	OUT_EV_HP => EV104,
	OUT_EV_LP => EV102,
(*	OUT_EV_LNK=> ,*)
	OUT_KEY   => KEY_PP2,
	OUT_THR   => THR_PP2
);
(*Link*)
EV107 := fbPP1.OUT_EV_LNK OR fbPP2.OUT_EV_LNK;  (******ANADIR si hace falta para la vibracion**************)

(*Alarms*)
Mute   := Mute   AND S101.AlLow AND S102.AlLow;
Bypass := Bypass AND (NOT S101.AlMax OR NOT S102.AlMax);
Buzzer := TANK.Enable AND (S101.AlHig OR S102.AlHig OR S101.AlMax OR S102.AlMax) AND NOT MUTE;

(*THROTTLE CALIBRATION*)
IF Calib1 THEN
	Calib2 := FALSE;

	CalThr := CalThr + CalInc;
	IF CalThr > CalMax THEN CalThr := CalMax; END_IF

	THR_PP1 := CalThr;
	THR_PP2 := 0.0;

	KEY_PP1 := TRUE;
	KEY_PP2 := TRUE;

	EV101 := FALSE;
	EV102 := FALSE;
	EV103 := FALSE;
	EV104 := FALSE;
ELSE
	CalThr := 0.0;
END_IF

IF Calib2 THEN
	Calib1 := FALSE;

	CalThr := CalThr + CalInc;
	IF CalThr > CalMax THEN CalThr := CalMax; END_IF

	THR_PP1 := 0.0;
	THR_PP2 := CalThr;

	KEY_PP1 := TRUE;
	KEY_PP2 := TRUE;

	EV101 := FALSE;
	EV102 := FALSE;
	EV103 := FALSE;
	EV104 := FALSE;
ELSE
	CalThr := 0.0;
END_IF
END_PROGRAM

(* POU FB/FB_POWERPACK, ST *)
FUNCTION_BLOCK FB_POWERPACK
VAR_INPUT
	Enable : BOOL;

	IN_HP : BOOL;
	IN_LP : BOOL;
END_VAR
VAR_IN_OUT
	HP_P : ST_SENSOR_BAR;
	LP_P : ST_SENSOR_BAR;
	CFG  : ST_POWERPACK_CFG;
END_VAR
VAR_OUTPUT
	OUT_EV_HP : BOOL;
	OUT_EV_LP : BOOL;
	OUT_EV_LNK: BOOL;
	OUT_KEY   : BOOL;
	OUT_THR   : REAL;
END_VAR
VAR
	State    : WORD;
	Hyst_Cnt : REAL;
	Hyst_ON  : BOOL;
	Thr_Cnt  : REAL;

END_VAR
IF NOT Enable THEN
	OUT_EV_HP  := FALSE;
	OUT_EV_LP  := FALSE;
	OUT_EV_LNK := FALSE;
	OUT_KEY    := FALSE;
	OUT_THR    := 0.0;

	State := 0;
	RETURN;
END_IF

IF LP_P.AlMax THEN IN_LP := FALSE; END_IF
IF HP_P.AlMax THEN IN_HP := FALSE; END_IF

CASE State OF
0: (*Init*)
	IF IN_LP AND IN_HP THEN
		OUT_EV_HP := TRUE;
		OUT_EV_LP := TRUE;
		OUT_EV_LNK:= FALSE;
		OUT_KEY   := TRUE;

		State := 30;

	ELSIF IN_LP THEN
		OUT_EV_HP := TRUE; (*Only LP Go with HP too*)
		OUT_EV_LP := TRUE;
		OUT_EV_LNK:= TRUE; (*Only LP Go with HP too*)
		OUT_KEY   := TRUE;

		Hyst_cnt := CFG.Hyst_TM + CFG.Cycle;
		State    := 10;

	ELSIF IN_HP THEN
		OUT_EV_HP := TRUE;
		OUT_EV_LP := FALSE;
		OUT_EV_LNK:= FALSE;
		OUT_KEY   := TRUE;

		State    := 20;

	ELSE
		OUT_EV_HP := FALSE;
		OUT_EV_LP := FALSE;
		OUT_EV_LNK:= FALSE;
		OUT_KEY   := FALSE;

	END_IF

	Thr_Cnt := 0.0;

10: (*LOW PRESS*)
	IF NOT IN_LP AND NOT IN_HP THEN
		OUT_EV_HP := FALSE;
		OUT_EV_LP := FALSE;
		OUT_EV_LNK:= FALSE;
		OUT_KEY   := FALSE;

		State := 0;

	ELSIF NOT IN_LP THEN (*Go to HP*)
		OUT_EV_HP := TRUE;
		OUT_EV_LP := FALSE;
		OUT_EV_LNK:= FALSE;

		State := 20;

	ELSIF IN_HP THEN
		OUT_EV_HP := TRUE;
		OUT_EV_LP := TRUE;
		OUT_EV_LNK:= FALSE;

		State := 30;

	ELSE
		IF Hyst_Cnt > CFG.Hyst_TM THEN
			Hyst_ON := TRUE;
		ELSE
			Hyst_ON  := FALSE;
			Hyst_Cnt := Hyst_Cnt + CFG.Cycle;
		END_IF

		IF LP_P.Bar > CFG.Hyst_HP AND Hyst_ON OR LP_P.Err THEN
			OUT_EV_HP  := FALSE;
			OUT_EV_LP  := TRUE;
			OUT_EV_LNK := FALSE;

			Hyst_cnt   := 0.0;

		ELSIF LP_P.Bar < CFG.Hyst_LP AND Hyst_ON THEN
			OUT_EV_HP  := TRUE; (*Only LP Go with HP too*)
			OUT_EV_LP  := TRUE;
			OUT_EV_LNK := TRUE; (*Only LP Go with HP too*)

			Hyst_cnt := 0.0;

		END_IF

	END_IF

20: (*HIGH PRESS*)
	IF NOT IN_LP AND NOT IN_HP THEN
		OUT_EV_HP := FALSE;
		OUT_EV_LP := FALSE;
		OUT_EV_LNK:= FALSE;
		OUT_KEY   := FALSE;

		State     := 0;

	ELSIF NOT IN_HP THEN
		OUT_EV_HP  := TRUE; (*Only LP Go with HP too*)
		OUT_EV_LP  := TRUE;
		OUT_EV_LNK := TRUE; (*Only LP Go with HP too*)

		Hyst_cnt := CFG.Hyst_TM + CFG.Cycle;
		State    := 10;

	ELSIF IN_LP THEN
		OUT_EV_HP := TRUE;
		OUT_EV_LP := TRUE;
		OUT_EV_LNK:= FALSE;

		State := 30;

	ELSE
		OUT_EV_HP := TRUE;
		OUT_EV_LP := FALSE;
		OUT_EV_LNK:= FALSE;

	END_IF

30: (*HP & LP*)
	IF NOT IN_LP AND NOT IN_HP THEN
		OUT_EV_HP := FALSE;
		OUT_EV_LP := FALSE;
		OUT_EV_LNK:= FALSE;
		OUT_KEY   := FALSE;

		State     := 0;

	ELSIF NOT IN_HP THEN (*Go to LP*)
		OUT_EV_HP  := TRUE; (*Only LP Go with HP too*)
		OUT_EV_LP  := TRUE;
		OUT_EV_LNK := TRUE; (*Only LP Go with HP too*)

		Hyst_cnt := CFG.Hyst_TM + CFG.Cycle;
		State    := 10;

	ELSIF NOT IN_LP THEN (*Go to HP*)
		OUT_EV_HP := TRUE;
		OUT_EV_LP := FALSE;
		OUT_EV_LNK:= FALSE;

		State := 20;

	ELSE
		OUT_EV_HP := TRUE;
		OUT_EV_LP := TRUE;
		OUT_EV_LNK:= FALSE;

	END_IF

END_CASE

IF OUT_KEY THEN
	IF Thr_Cnt > 0.2 THEN
		IF OUT_EV_HP AND OUT_EV_LP THEN
			OUT_Thr := MAX(CFG.Thr_HP,CFG.Thr_LP);
		ELSIF OUT_EV_LP THEN
			OUT_Thr := CFG.Thr_LP;
		ELSE
			OUT_Thr := CFG.Thr_HP;
		END_IF

	ELSE
		Thr_Cnt := Thr_Cnt + CFG.Cycle;
		OUT_Thr := 0.0;
	END_IF

ELSE
	OUT_THR := 0.0;

END_IF
END_FUNCTION_BLOCK

(* POU TOFARO, ST *)
PROGRAM TOFARO
VAR CONSTANT
	UDP_BUF_SIZE  : WORD := 4096;

END_VAR
VAR
	fbUdpSend        : FB_UDP_SEND;
	fbUdpRecv        : FB_UDP_RECV;
	fbSocketCloseAll : FB_SocketCloseAll;
    bCloseAll 	     : BOOL := TRUE;

	Send_Id          : DWORD;
	Send_NumberOfVars: WORD;
	Send_Offset      : WORD;
	Send_Buffer      : ARRAY[0..UDP_BUF_SIZE] OF BYTE;

	AuxVar : REAL;

	Recv_Id          : DWORD;
	Recv_NumberOfVars: WORD;
	Recv_Offset      : WORD;
	Recv_Buffer      : ARRAY[0..UDP_BUF_SIZE] OF BYTE;
	Recv_ToggleOLD   : BOOL;
	Recv_OldId       : DWORD;
	NoRecv_Cnt       : REAL;
	Recv_Live        : BOOL;

	rBar1 : REAL;
	rBar2 : REAL;
	rHeel : REAL;

	rRunP : REAL;
	rPriP : REAL;
	rMain : REAL;
	rRunS : REAL;
	rPriS : REAL;
	rSecP : REAL;
	rSecS : REAL;



END_VAR
(*UDP STREAMING*)
IF bCloseAll THEN (*On PLC reset or program download close all old connections *)
	bCloseAll := FALSE;
	fbUdpSend( bEnable:= FALSE );
	fbSocketCloseAll( bExecute:= TRUE, tTimeout:= T#10s );

	Recv_Live := FALSE;
ELSE
	fbSocketCloseAll( bExecute:= FALSE );
END_IF

IF NOT fbSocketCloseAll.bBusy THEN

(* UDP Inputs *)
	fbUdpRecv(
		bEnable    := TRUE,
		nLocalPort := PARAMS.nUDPRecvPort,
		pBuffer    := ADR(Recv_Buffer),
		wBufLen    := UDP_BUF_SIZE,
	);

	IF fbUdpRecv.bRecToggle <> Recv_ToggleOLD THEN
		Recv_ToggleOLD := fbUdpRecv.bRecToggle;

		IF fbUdpRecv.nRecBytes >= 48 THEN (* 10*4 + 8 Check size*)
			MEMCPY( ADR(Recv_Id          ), ADR(Recv_Buffer[0]), 4);
			MEMCPY( ADR(Recv_NumberOfVars), ADR(Recv_Buffer[4]), 2);
			MEMCPY( ADR(Recv_Offset      ), ADR(Recv_Buffer[6]), 2);

			(* 1*) MEMCPY( ADR(rBar1) , ADR(Recv_Buffer[ 8]), 4);
			(* 2*) MEMCPY( ADR(rBar2) , ADR(Recv_Buffer[12]), 4);
			(* 3*) MEMCPY( ADR(rHeel) , ADR(Recv_Buffer[16]), 4);
			(* 4*) MEMCPY( ADR(rRunP) , ADR(Recv_Buffer[20]), 4);
			(* 5*) MEMCPY( ADR(rPriP) , ADR(Recv_Buffer[24]), 4);
			(* 6*) MEMCPY( ADR(rMain) , ADR(Recv_Buffer[28]), 4);
			(* 7*) MEMCPY( ADR(rRunS) , ADR(Recv_Buffer[32]), 4);
			(* 8*) MEMCPY( ADR(rPriS) , ADR(Recv_Buffer[36]), 4);
			(* 9*) MEMCPY( ADR(rSecP) , ADR(Recv_Buffer[40]), 4);
			(*10*) MEMCPY( ADR(rSecS) , ADR(Recv_Buffer[44]), 4);

		END_IF
	END_IF

	IF Recv_Id <> Recv_OldId THEN
		NoRecv_Cnt := 0;
		Recv_OldId := Recv_Id;
		Recv_Live  := TRUE;
	ELSE
		NoRecv_Cnt := NoRecv_Cnt + MAIN.Cycle_Time;
	END_IF

	IF NoRecv_Cnt > 1 THEN
		Recv_Live := FALSE;
	END_IF

	IF NoRecv_Cnt > 10 THEN
		bCloseAll  := TRUE;
		NoRecv_Cnt := 0;
	END_IF

(*UDP Outputs*)
	IF fbUdpSend.eStep = UDP_STATE_SEND_START AND PARAMS.nUDPSendTime > 0 THEN

		(*Press Sensors*)
		(* 1*)MEMCPY( ADR(Send_Buffer[  8]), ADR(  P010.Bar ), 4); (*Tank*)
		(* 2*)MEMCPY( ADR(Send_Buffer[ 12]), ADR(  P101.Bar ), 4); (*PowerPack Low Press. Line*)
		(* 3*)MEMCPY( ADR(Send_Buffer[ 16]), ADR(  P103.Bar ), 4); (*Main High Press. Line*)
		(* 4*)MEMCPY( ADR(Send_Buffer[ 20]), ADR(  P201.Bar ), 4); (*Main Low Press. Line*)

		(* 5*)MEMCPY( ADR(Send_Buffer[ 24]), ADR(  P301.Bar ), 4); (*A3 Tack*)
		(* 6*)MEMCPY( ADR(Send_Buffer[ 28]), ADR(  P303.Bar ), 4); (*FRO Tack*)
		(* 7*)MEMCPY( ADR(Send_Buffer[ 32]), ADR(  P305.Bar ), 4); (*J5*)
		(* 8*)MEMCPY( ADR(Send_Buffer[ 36]), ADR(  P307.Bar ), 4); (*J4*)
		(* 9*)MEMCPY( ADR(Send_Buffer[ 40]), ADR(  P309.Bar ), 4); (*Forastay*)
		(*10*)MEMCPY( ADR(Send_Buffer[ 44]), ADR(  P311.Bar ), 4); (*J2*)

		(*11*)MEMCPY( ADR(Send_Buffer[ 48]), ADR(  P501.Bar ), 4); (*Jib InOut*)
		(*12*)MEMCPY( ADR(Send_Buffer[ 52]), ADR(  P503.Bar ), 4); (*Jib UpDw*)
		(*13*)MEMCPY( ADR(Send_Buffer[ 56]), ADR(  P505.Bar ), 4); (*Vang*)

		(*14*)MEMCPY( ADR(Send_Buffer[ 60]), ADR(  P601.Bar ), 4); (*Propulsion Dw*)
		(*15*)MEMCPY( ADR(Send_Buffer[ 64]), ADR(  P603.Bar ), 4); (*Propulsion Up*)
		(*16*)MEMCPY( ADR(Send_Buffer[ 68]), ADR(  P605.Bar ), 4); (*Trim Tab Out*)
		(*17*)MEMCPY( ADR(Send_Buffer[ 72]), ADR(  P607.Bar ), 4); (*Trim Tab In*)

		(*18*)MEMCPY( ADR(Send_Buffer[ 76]), ADR(  P701.Bar ), 4); (*Inner Staysail*)
		(*19*)MEMCPY( ADR(Send_Buffer[ 80]), ADR(  P703.Bar ), 4); (*Outhau*)
		(*20*)MEMCPY( ADR(Send_Buffer[ 84]), ADR(  P705.Bar ), 4); (*Main Cunningham*)
		(*21*)MEMCPY( ADR(Send_Buffer[ 88]), ADR(  P707.Bar ), 4); (*Bottom Deflectorl*)
		(*22*)MEMCPY( ADR(Send_Buffer[ 92]), ADR(  P709.Bar ), 4); (*Top Deflector*)

		(*23*)MEMCPY( ADR(Send_Buffer[ 96]), ADR(  P802.Bar ), 4); (*Daggerborad Port Pump*)
		(*24*)MEMCPY( ADR(Send_Buffer[100]), ADR(  P804.Bar ), 4); (*Daggerborad Stbd Pump*)

		(*25*)MEMCPY( ADR(Send_Buffer[104]), ADR(  P901.Bar ), 4); (*Backstay Tail Port*)
		(*26*)MEMCPY( ADR(Send_Buffer[108]), ADR(  P903.Bar ), 4); (*Backstay Tail Stbd*)

		(*27*)MEMCPY( ADR(Send_Buffer[112]), ADR( P1001.Bar ), 4); (*Keel IN*)
		(*28*)MEMCPY( ADR(Send_Buffer[116]), ADR( P1002.Bar ), 4); (*Keel OUT*)

		(*29*)MEMCPY( ADR(Send_Buffer[120]), ADR( P1101.Bar ), 4); (*Propulsion*)
		(*30*)MEMCPY( ADR(Send_Buffer[124]), ADR( P1102.Bar ), 4); (*Propulsion*)

		(*31*)MEMCPY( ADR(Send_Buffer[128]), ADR( P1202.Bar ), 4); (*Primary Winch Stbd A*)
		(*32*)MEMCPY( ADR(Send_Buffer[132]), ADR( P1203.Bar ), 4); (*Primary Winch Stbd B*)
		(*33*)MEMCPY( ADR(Send_Buffer[136]), ADR( P1204.Bar ), 4); (*Pit Winch Stbd A*)
		(*34*)MEMCPY( ADR(Send_Buffer[140]), ADR( P1205.Bar ), 4); (*Pit Winch Stbd B*)
		(*35*)MEMCPY( ADR(Send_Buffer[144]), ADR( P1206.Bar ), 4); (*Mainsheet Winch A*)
		(*36*)MEMCPY( ADR(Send_Buffer[148]), ADR( P1207.Bar ), 4); (*Mainsheet Winch B*)
		(*37*)MEMCPY( ADR(Send_Buffer[152]), ADR( P1208.Bar ), 4); (*Runner Winch Port A*)
		(*38*)MEMCPY( ADR(Send_Buffer[156]), ADR( P1209.Bar ), 4); (*Runner Winch Port B*)
		(*39*)MEMCPY( ADR(Send_Buffer[160]), ADR( P1210.Bar ), 4); (*Primary Winch Port A*)
		(*40*)MEMCPY( ADR(Send_Buffer[164]), ADR( P1211.Bar ), 4); (*Primary Winch Port B*)
		(*41*)MEMCPY( ADR(Send_Buffer[168]), ADR( P1212.Bar ), 4); (*Secondary Winch Port A*)
		(*42*)MEMCPY( ADR(Send_Buffer[172]), ADR( P1213.Bar ), 4); (*Secondary Winch Port B*)
		(*43*)MEMCPY( ADR(Send_Buffer[176]), ADR( P1214.Bar ), 4); (*Pit Winch Port	A*)
		(*44*)MEMCPY( ADR(Send_Buffer[180]), ADR( P1215.Bar ), 4); (*Pit Winch Port	B*)
		(*45*)MEMCPY( ADR(Send_Buffer[184]), ADR( P1216.Bar ), 4); (*Daggerborad Port Ease*)
		(*46*)MEMCPY( ADR(Send_Buffer[188]), ADR( P1219.Bar ), 4); (*Daggerborad Stbd Ease*)

		(*47*)MEMCPY( ADR(Send_Buffer[192]), ADR( P1301.Bar ), 4); (*Traveller A*)
		(*48*)MEMCPY( ADR(Send_Buffer[196]), ADR( P1302.Bar ), 4); (*Traveller B*)

		(*49*)MEMCPY( ADR(Send_Buffer[200]), ADR( P1602.Bar ), 4); (*Runner Winch Stbd A*)
		(*50*)MEMCPY( ADR(Send_Buffer[204]), ADR( P1603.Bar ), 4); (*Runner Winch Stbd B*)
		(*51*)MEMCPY( ADR(Send_Buffer[208]), ADR( P1604.Bar ), 4); (*Secondary Winch Stbd A*)
		(*52*)MEMCPY( ADR(Send_Buffer[212]), ADR( P1605.Bar ), 4); (*Secondary Winch Stbd B*)

		(*Position Sensors*)
		(*53*)MEMCPY( ADR(Send_Buffer[216]), ADR(  LS301.Pos ), 4); (*A3 Tack*)
		(*54*)MEMCPY( ADR(Send_Buffer[220]), ADR(  LS303.Pos ), 4); (*FRO Tack*)
		(*55*)MEMCPY( ADR(Send_Buffer[224]), ADR(  LS305.Pos ), 4); (*J5*)
		(*56*)MEMCPY( ADR(Send_Buffer[228]), ADR(  LS307.Pos ), 4); (*J4*)
		(*57*)MEMCPY( ADR(Send_Buffer[232]), ADR(  LS309.Pos ), 4); (*Forastay*)
		(*58*)MEMCPY( ADR(Send_Buffer[236]), ADR(  LS311.Pos ), 4); (*J2*)

		(*59*)MEMCPY( ADR(Send_Buffer[240]), ADR(  LS601.Pos ), 4); (*Propulsion*)
		(*60*)MEMCPY( ADR(Send_Buffer[244]), ADR(  LS605.Pos ), 4); (*Trim Tab*)

		(*61*)MEMCPY( ADR(Send_Buffer[248]), ADR(  LS707.Pos ), 4); (*Bottom Deflector*)
		(*62*)MEMCPY( ADR(Send_Buffer[252]), ADR(  LS709.Pos ), 4); (*Top Deflector*)

		(*63*)MEMCPY( ADR(Send_Buffer[256]), ADR(  LS801.Pos ), 4); (*Daggerboard Port*)
		(*64*)MEMCPY( ADR(Send_Buffer[260]), ADR(  LS803.Pos ), 4); (*Daggerboard Stbd*)

		(*65*)MEMCPY( ADR(Send_Buffer[264]), ADR(  LS901.Pos ), 4); (*Backstay Tail Port*)
		(*66*)MEMCPY( ADR(Send_Buffer[268]), ADR(  LS903.Pos ), 4); (*Backstay Tail Stbd*)

		(*67*)MEMCPY( ADR(Send_Buffer[272]), ADR( LS1001.Pos ), 4); (*Keel Main*)
		(*68*)MEMCPY( ADR(Send_Buffer[276]), ADR( LS1002.Pos ), 4); (*Keel Recovery*)

		(*69*)MEMCPY( ADR(Send_Buffer[280]), ADR( LS1303.Pos ), 4); (*Traveller*)

		(*Water Ballast*)
		(*70*)MEMCPY( ADR(Send_Buffer[284]), ADR( LS021.Pos ), 4); (*Aft. Tank (Port)*)
		(*71*)MEMCPY( ADR(Send_Buffer[288]), ADR( LS022.Pos ), 4); (*Fwd. Tank (Port)*)
		(*72*)MEMCPY( ADR(Send_Buffer[292]), ADR( LS023.Pos ), 4); (*Aft. Tank (Stbd)*)
		(*73*)MEMCPY( ADR(Send_Buffer[296]), ADR( LS024.Pos ), 4); (*Fwd. Tank (Stbd)*)

		(*Engine*)
		(*74*)MEMCPY( ADR(Send_Buffer[300]), ADR( RECV_J1939.F004.EngineActualSpeed        ), 4); (*Engine Speed RPM*)
			  AuxVar := SINT_TO_REAL( RECV_J1939.F004.EngineActualTorque );
		(*75*)MEMCPY( ADR(Send_Buffer[304]), ADR( AuxVar                                   ), 4); (*Engine Torque %*)
		(*76*)MEMCPY( ADR(Send_Buffer[308]), ADR( RECV_J1939.FEEE.EngineCoolantTemperature ), 4); (*Engine Coolant Temp*)
		(*77*)MEMCPY( ADR(Send_Buffer[312]), ADR( RECV_J1939.FEEF.EngineOilPressure        ), 4); (*Engine Oil Press kPa*)
		(*78*)MEMCPY( ADR(Send_Buffer[316]), ADR( Prop_RPM                                 ), 4); (*Propulsion RPM*)

		(*Tank*)
		(*79*)MEMCPY( ADR(Send_Buffer[320]), ADR( S011.Deg ), 4); (*Oil Tank Temp*)

			  IF    MAIN.fbBowThrUpDw.IN_SF1 THEN AuxVar :=   0.0;
			  ELSIF MAIN.fbBowThrUpDw.IN_SF2 THEN AuxVar := 100.0;
			  ELSE                                AuxVar :=  50.0;
			  END_IF

		(*80*)MEMCPY( ADR(Send_Buffer[324]), ADR( AuxVar ), 4); (*BowThrUpDw*)

		(*HP VALVES*)
		(*81*)MEMCPY( ADR(Send_Buffer[328]), ADR( MAIN.fbSE301.ToFaroValue ), 4);
		(*82*)MEMCPY( ADR(Send_Buffer[332]), ADR( MAIN.fbSE303.ToFaroValue ), 4);
		(*83*)MEMCPY( ADR(Send_Buffer[336]), ADR( MAIN.fbSE305.ToFaroValue ), 4);
		(*84*)MEMCPY( ADR(Send_Buffer[340]), ADR( MAIN.fbSE307.ToFaroValue ), 4);
		(*85*)MEMCPY( ADR(Send_Buffer[344]), ADR( MAIN.fbSE309.ToFaroValue ), 4);
		(*86*)MEMCPY( ADR(Send_Buffer[348]), ADR( MAIN.fbSE311.ToFaroValue ), 4);

		(*87*)MEMCPY( ADR(Send_Buffer[352]), ADR( MAIN.fbSE501.ToFaroValue ), 4);
		(*88*)MEMCPY( ADR(Send_Buffer[356]), ADR( MAIN.fbSE503.ToFaroValue ), 4);
		(*89*)MEMCPY( ADR(Send_Buffer[360]), ADR( MAIN.fbSE505.ToFaroValue ), 4);

		(*90*)MEMCPY( ADR(Send_Buffer[364]), ADR( MAIN.fbDE601.ToFaroValue ), 4);
		(*91*)MEMCPY( ADR(Send_Buffer[368]), ADR( MAIN.fbDE605.ToFaroValue ), 4);

		(*92*)MEMCPY( ADR(Send_Buffer[372]), ADR( MAIN.fbSE701.ToFaroValue ), 4);
		(*93*)MEMCPY( ADR(Send_Buffer[376]), ADR( MAIN.fbSE703.ToFaroValue ), 4);
		(*94*)MEMCPY( ADR(Send_Buffer[380]), ADR( MAIN.fbSE705.ToFaroValue ), 4);
		(*95*)MEMCPY( ADR(Send_Buffer[384]), ADR( MAIN.fbSE707.ToFaroValue ), 4);
		(*96*)MEMCPY( ADR(Send_Buffer[388]), ADR( MAIN.fbSE709.ToFaroValue ), 4);

		(*97*)MEMCPY( ADR(Send_Buffer[392]), ADR( MAIN.fbBSY.ToFaroValueP ), 4);
		(*98*)MEMCPY( ADR(Send_Buffer[396]), ADR( MAIN.fbBSY.ToFaroValueS ), 4);

		(*99*)MEMCPY( ADR(Send_Buffer[400]), ADR( MAIN.fbTraveller.ToFaroValue ), 4);

		(*LP VALVES*)
		(*100*)AuxVar := UINT_TO_REAL(EVP001); MEMCPY( ADR(Send_Buffer[404]), ADR( AuxVar ), 4);
		(*101*)AuxVar := UINT_TO_REAL(EVP002); MEMCPY( ADR(Send_Buffer[408]), ADR( AuxVar ), 4);

		(*102*)AuxVar := INT_TO_REAL(EVP1202_3); MEMCPY( ADR(Send_Buffer[412]), ADR( AuxVar ), 4);
		(*103*)AuxVar := INT_TO_REAL(EVP1204_5); MEMCPY( ADR(Send_Buffer[416]), ADR( AuxVar ), 4);
		(*104*)AuxVar := INT_TO_REAL(EVP1206_7); MEMCPY( ADR(Send_Buffer[420]), ADR( AuxVar ), 4);
		(*105*)AuxVar := INT_TO_REAL(EVP1208_9); MEMCPY( ADR(Send_Buffer[424]), ADR( AuxVar ), 4);
		(*106*)AuxVar := INT_TO_REAL(EVP1210_1); MEMCPY( ADR(Send_Buffer[428]), ADR( AuxVar ), 4);
		(*107*)AuxVar := INT_TO_REAL(EVP1212_3); MEMCPY( ADR(Send_Buffer[432]), ADR( AuxVar ), 4);
		(*108*)AuxVar := INT_TO_REAL(EVP1214_5); MEMCPY( ADR(Send_Buffer[436]), ADR( AuxVar ), 4);
		(*109*)AuxVar := INT_TO_REAL(EVP1216_7); MEMCPY( ADR(Send_Buffer[440]), ADR( AuxVar ), 4);
		(*110*)AuxVar := INT_TO_REAL(EVP1218_9); MEMCPY( ADR(Send_Buffer[444]), ADR( AuxVar ), 4);
		(*111*)AuxVar := INT_TO_REAL(EVP1220_1); MEMCPY( ADR(Send_Buffer[448]), ADR( AuxVar ), 4);

		(*112*)AuxVar := INT_TO_REAL(EVP402_3); MEMCPY( ADR(Send_Buffer[452]), ADR( AuxVar ), 4);
		(*113*)AuxVar := INT_TO_REAL(EVP404_5); MEMCPY( ADR(Send_Buffer[456]), ADR( AuxVar ), 4);
		(*114*)AuxVar := INT_TO_REAL(EVP406_7); MEMCPY( ADR(Send_Buffer[460]), ADR( AuxVar ), 4);

		(*115*)AuxVar := INT_TO_REAL(EVP1602_3); MEMCPY( ADR(Send_Buffer[464]), ADR( AuxVar ), 4);
		(*116*)AuxVar := INT_TO_REAL(EVP1604_5); MEMCPY( ADR(Send_Buffer[468]), ADR( AuxVar ), 4);
		(*117*)AuxVar := INT_TO_REAL(EVP1606_7); MEMCPY( ADR(Send_Buffer[472]), ADR( AuxVar ), 4);
		(*118*)AuxVar := INT_TO_REAL(EVP1608_9); MEMCPY( ADR(Send_Buffer[476]), ADR( AuxVar ), 4);
		(*119*)AuxVar := INT_TO_REAL(EVP1610_1); MEMCPY( ADR(Send_Buffer[480]), ADR( AuxVar ), 4);

		(*FUNCTIONS IN USE*)
		(*120*)AuxVar := UINT_TO_REAL(POWERPACK.NHP); MEMCPY( ADR(Send_Buffer[484]), ADR( AuxVar ), 4);
		(*121*)AuxVar := UINT_TO_REAL(POWERPACK.NLP); MEMCPY( ADR(Send_Buffer[488]), ADR( AuxVar ), 4);
		(*122*)AuxVar := UINT_TO_REAL(POWERPACK.NW ); MEMCPY( ADR(Send_Buffer[492]), ADR( AuxVar ), 4);

		(*123*)MEMCPY( ADR(Send_Buffer[496]), ADR( POWERPACK.LP_Perc ), 4); (*Flow Percentage*)

		(*WINCHES INPUTS*)
		(*124*)MEMCPY( ADR(Send_Buffer[500]), ADR( MAIN.fbW1202.ToFaroInput ), 4); (*Primary Winch Stbd*)
		(*125*)MEMCPY( ADR(Send_Buffer[504]), ADR( MAIN.fbW1204.ToFaroInput ), 4); (*Pit Winch Stbd*)
		(*126*)MEMCPY( ADR(Send_Buffer[508]), ADR( MAIN.fbW1206.ToFaroInput ), 4); (*Mainsheet Winch*)
		(*127*)MEMCPY( ADR(Send_Buffer[512]), ADR( MAIN.fbW1208.ToFaroInput ), 4); (*Runner Winch Port*)
		(*128*)MEMCPY( ADR(Send_Buffer[516]), ADR( MAIN.fbW1210.ToFaroInput ), 4); (*Primary Winch Port*)
		(*129*)MEMCPY( ADR(Send_Buffer[520]), ADR( MAIN.fbW1212.ToFaroInput ), 4); (*Secondary Winch Port*)
		(*130*)MEMCPY( ADR(Send_Buffer[524]), ADR( MAIN.fbW1214.ToFaroInput ), 4); (*Pit Winch Port*)

		(*131*)MEMCPY( ADR(Send_Buffer[528]), ADR( MAIN.fbW1602.ToFaroInput ), 4); (*Runner Winch Stbd*)
		(*132*)MEMCPY( ADR(Send_Buffer[532]), ADR( MAIN.fbW1604.ToFaroInput ), 4); (*Secondary Winch Stbd*)

		(*WINCHES OUTPUS*)
		(*133*)MEMCPY( ADR(Send_Buffer[536]), ADR( MAIN.fbW1202.ToFaroOutput ), 4); (*Primary Winch Stbd*)
		(*134*)MEMCPY( ADR(Send_Buffer[540]), ADR( MAIN.fbW1204.ToFaroOutput ), 4); (*Pit Winch Stbd*)
		(*135*)MEMCPY( ADR(Send_Buffer[544]), ADR( MAIN.fbW1206.ToFaroOutput ), 4); (*Mainsheet Winch*)
		(*136*)MEMCPY( ADR(Send_Buffer[548]), ADR( MAIN.fbW1208.ToFaroOutput ), 4); (*Runner Winch Port*)
		(*137*)MEMCPY( ADR(Send_Buffer[552]), ADR( MAIN.fbW1210.ToFaroOutput ), 4); (*Primary Winch Port*)
		(*138*)MEMCPY( ADR(Send_Buffer[556]), ADR( MAIN.fbW1212.ToFaroOutput ), 4); (*Secondary Winch Port*)
		(*139*)MEMCPY( ADR(Send_Buffer[560]), ADR( MAIN.fbW1214.ToFaroOutput ), 4); (*Pit Winch Port*)

		(*140*)MEMCPY( ADR(Send_Buffer[564]), ADR( MAIN.fbW1602.ToFaroOutput ), 4); (*Runner Winch Stbd*)
		(*141*)MEMCPY( ADR(Send_Buffer[568]), ADR( MAIN.fbW1604.ToFaroOutput ), 4); (*Secondary Winch Stbd*)

		(*Extra Variables*)
		(*142*)AuxVar := UINT_TO_REAL(MAIN.fbMastSetup.Selected_MS); MEMCPY( ADR(Send_Buffer[572]), ADR( AuxVar ), 4);
		(*143*)AuxVar := UINT_TO_REAL(MAIN.fbMastSetup.Selected_HS); MEMCPY( ADR(Send_Buffer[576]), ADR( AuxVar ), 4);

		(*144*)MEMCPY( ADR(Send_Buffer[580]), ADR( S1100.Deg ), 4);

		(*145*)MEMCPY( ADR(Send_Buffer[584]), ADR( ENGINE.fbEngine.Engine_RPM), 4); (*TargetRPM*)
		(*146*)MEMCPY( ADR(Send_Buffer[588]), ADR( SEND_J1939.PedalPerc), 4); (*TagetRPM_Perc*)

		(*147*)MEMCPY( ADR(Send_Buffer[592]), ADR( P003.Bar ), 4); (*TagetRPM_Perc*)

(*
*)

		Send_ID           := Send_ID + 1;
		Send_NumberOfVars := 147;
		Send_Offset       := 0;

		MEMCPY( ADR(Send_Buffer[ 0]), ADR(Send_Id           ), 4);
		MEMCPY( ADR(Send_Buffer[ 4]), ADR(Send_NumberOfVars ), 2);
		MEMCPY( ADR(Send_Buffer[ 6]), ADR(Send_Offset       ), 2);

	END_IF

	fbUdpSend(
		bEnable    := PARAMS.nUDPSendTime > 0,
		sRemoteHost:= PARAMS.sUDPSendHost,
		nRemotePort:= PARAMS.nUDPSendPort,
		nTime      := PARAMS.nUDPSendTime,

		pBuffer:= ADR(Send_Buffer),
		wBufLen:= 596, (*8 + 147*4*)
		nCycle := 20,
	);

END_IF
END_PROGRAM

(* POU SEND_J1939, ST *)
PROGRAM SEND_J1939
VAR
	i: INT;
	iToSend  : INT;
	aTxFrame : ARRAY [0..9] OF VARTYPE_EXTCANQUEUE;

	fbFF70 : FB_CODE_FF70;

	PedalPerc  : REAL;
	PedalFault : BOOL;
END_VAR
(*2800 = 100%*)
PedalPerc  := ENGINE.fbEngine.Engine_RPM * 0.04504504505 - 30.63063063; (*NEW*)
(*PedalPerc  := ENGINE.fbEngine.Engine_RPM * 0.0448 - 31.883;*)
(*PedalFault := NOT fbEngine.Enable;*)

(*Engine Pedal frame*)
fbFF70(
	Enable := ENGINE.fbEngine.Enable,
	Source     := 16#10,
	PedalPerc  := PedalPerc,
	PedalID    := 0,
	PedalFault := PedalFault,

	TaskTime     := 5,
	TransmitTime := 50
);

IF fbFF70.OUT_Enable THEN
	IF iToSend < 10 THEN
		aTxFrame[iToSend] := fbFF70.OUT;
		iToSend := iToSend + 1;
	END_IF
END_IF

(*SendingCAN*)
IF J1939_Outputs.TxCounter = J1939_Inputs.TxCounter AND iToSend > 0 THEN
	FOR i := 0 TO iToSend-1 BY 1 DO
		MEMCPY( destAddr := ADR(J1939_Outputs.TxMessages[i] ), srcAddr := ADR(aTxFrame[i].length), n := 14 );
	END_FOR

	J1939_Outputs.NoOfTxMessages := iToSend;
	J1939_Outputs.TxCounter      := J1939_Outputs.TxCounter + 1;

	iToSend := 0;
END_IF
END_PROGRAM

(* POU PGN FB/FB_CODE_FF70, ST *)
FUNCTION_BLOCK FB_CODE_FF70 (*Torque / Speed Control*)
VAR_INPUT
	Enable   : BOOL;
	Source   : BYTE := 16#10;
	Priority : BYTE := 16#02;

	TaskTime     : WORD; (*PLC Taks Time (ms) eg: 10ms*)
	TransmitTime : WORD; (*Synchronous Transmision Time (ms) eg: 50ms*)

	PedalPerc  : REAL;
	PedalID    : BYTE;
	PedalFault : BOOL;
END_VAR
VAR_OUTPUT
	OUT : VARTYPE_EXTCANQUEUE;
	OUT_Enable : BOOL;
END_VAR
VAR
	TimeCnt : WORD;
	dwSrc   : DWORD;
	dwPty   : DWORD;

	bySpeedCtrl  : BYTE;
	byTorqueCtrl : BYTE;
END_VAR
IF Enable THEN
	TimeCnt := TimeCnt + TaskTime;

	IF TransmitTime <= TimeCnt THEN
		TimeCnt := 0;
		dwSrc   := Source;
		dwPty   := Priority AND 16#07;
		dwPty   := SHL( dwPty, 26 );

		REAL_TO_BUFFER( pBuffer:= ADR(OUT.rxData[0]), ByteSize := 2, Value:= PedalPerc, Scale:= 0.1, Offset := 0.0 );

		OUT.rxData[2] := PedalID;
		OUT.rxData[3] := 16#00;
		OUT.rxData[3].0 := PedalFault;
		OUT.rxData[4] := 16#00;
		OUT.rxData[5] := 16#00;
		OUT.rxData[6] := 16#00;
		OUT.rxData[7] := 16#00;

		OUT.length := 8;
		Out.cobId  := 16#80FF7000 OR dwSrc OR dwPty;
		OUT_Enable := TRUE;
	ELSE
		OUT_Enable := FALSE;

	END_IF
ELSE
	Out_Enable := FALSE;

END_IF
END_FUNCTION_BLOCK

(* POU FUN/F_CALC_SENSOR_NC, ST *)
FUNCTION F_CALC_SENSOR_NC : BOOL
VAR_INPUT
	IN    : BOOL;
	Clear : BOOL;
	Cycle : REAL;
	Delay : REAL;
END_VAR
VAR_IN_OUT
	Sensor : ST_SENSOR_SWITCH;
END_VAR
VAR
END_VAR
IF Clear THEN
	Sensor.Alarm.Alarm := FALSE;
	Sensor.Alarm.Adver := FALSE;
	Sensor.Alarm.AlCnt := 0;
	Sensor.Alarm.AlLen := 0.0;
END_IF

IF NOT IN THEN
	IF Sensor.Count >= Delay THEN
		IF NOT Sensor.Alarm.Alarm THEN
			Sensor.Alarm.AlCnt  := Sensor.Alarm.AlCnt + 1;
			Sensor.Alarm.AlLen  := 0.0;
			Sensor.Alarm.TimeInit := INPUTS.sLocal;
			Sensor.Alarm.AlInit   := TRUE;

			Sensor.Alarm.Text   := Sensor.Desc;

		ELSE
			Sensor.Alarm.AlLen  := Sensor.Alarm.AlLen + MAIN.Cycle_Time;

		END_IF

		Sensor.Alarm.Adver := TRUE;
		Sensor.Alarm.Alarm := TRUE;

	ELSE
		Sensor.Count := Sensor.Count + Cycle;

	END_IF

ELSE
	IF Sensor.Alarm.Alarm THEN
		Sensor.Alarm.TimeEnd := INPUTS.sLocal;
		Sensor.Alarm.AlEnd   := TRUE;

	END_IF

	Sensor.Alarm.Alarm := FALSE;
	Sensor.Count       := 0;
END_IF
END_FUNCTION

(* POU FUN/F_CALC_SENSOR_BAR, ST *)
FUNCTION F_CALC_SENSOR_BAR : BOOL
VAR_INPUT
	IN    : REAL;
	Clear : BOOL;
END_VAR
VAR_IN_OUT
	Sensor : ST_SENSOR_BAR;
END_VAR
VAR
END_VAR
(*AVG*)
IF Sensor.Avg_Pos > 4 THEN Sensor.Avg_Pos := 0; END_IF

Sensor.Avg_Sum := Sensor.Avg_Sum + IN - Sensor.Avg_Buf[Sensor.Avg_Pos];
Sensor.Avg_Buf[Sensor.Avg_Pos] := IN;
Sensor.Avg_Pos := Sensor.Avg_Pos + 1;

Sensor.Raw := Sensor.Avg_Sum / 5.0;
Sensor.Err := Sensor.Raw < Sensor.MinRaw OR Sensor.Raw > Sensor.MaxRaw;

(*CALIB*)
Sensor.Bar := Sensor.Raw * Sensor.Cal_K + Sensor.Cal_Off;

(*ALARM*)
IF Clear THEN
	Sensor.Alarm.Alarm := FALSE;
	Sensor.Alarm.Adver := FALSE;
	Sensor.Alarm.AlCnt := 0;
	Sensor.Alarm.AlLen := 0.0;
(*	Sensor.AdverVal    := Sensor.Bar;*) (*Lo reseteo *)

END_IF

IF Sensor.Err THEN
	IF NOT Sensor.Alarm.Alarm OR NOT Sensor.AlErr THEN
		Sensor.Alarm.AlCnt  := Sensor.Alarm.AlCnt + 1;
		Sensor.Alarm.AlLen  := 0.0;
		Sensor.Alarm.TimeInit := INPUTS.sLocal;
		Sensor.Alarm.AlInit   := TRUE;

		Sensor.Alarm.Text := CONCAT( Sensor.Desc, ' Press. Sensor Broken/Disconnected.' );

	ELSE
		Sensor.Alarm.AlLen  := Sensor.Alarm.AlLen + MAIN.Cycle_Time;

	END_IF

	Sensor.Alarm.Alarm := TRUE;
	Sensor.Alarm.Adver := TRUE;

	Sensor.AlErr    := TRUE;
	Sensor.AlMax    := FALSE;
	Sensor.AlMin    := FALSE;
	Sensor.AdverVal := 0.0;

ELSIF Sensor.MaxBar > 0 AND Sensor.Bar > Sensor.MaxBar THEN
	IF NOT Sensor.Alarm.Alarm OR NOT Sensor.AlMax THEN
		Sensor.Alarm.AlCnt  := Sensor.Alarm.AlCnt + 1;
		Sensor.Alarm.AlLen  := 0.0;
		Sensor.Alarm.TimeInit := INPUTS.sLocal;
		Sensor.Alarm.AlInit   := TRUE;

		Sensor.AdverVal     := Sensor.Bar;
	ELSE
		Sensor.Alarm.AlLen  := Sensor.Alarm.AlLen + MAIN.Cycle_Time;
	END_IF

	Sensor.Alarm.Alarm := TRUE;
	Sensor.Alarm.Adver := TRUE;

	Sensor.AlErr    := FALSE;
	Sensor.AlMax    := TRUE;
	Sensor.AlMin    := FALSE;
 	Sensor.AdverVal := MAX( Sensor.Bar, Sensor.AdverVal );

	Sensor.Alarm.Text := CONCAT( Sensor.Desc      , ' Overpressured: ' );
	Sensor.Alarm.Text := CONCAT( Sensor.Alarm.Text, REAL_TO_STRING(Sensor.AdverVal) );

ELSIF Sensor.MinBar > 0 AND Sensor.Bar < Sensor.MinBar THEN
	IF NOT Sensor.Alarm.Alarm OR NOT Sensor.AlMin THEN
		Sensor.Alarm.AlCnt  := Sensor.Alarm.AlCnt + 1;
		Sensor.Alarm.AlLen  := 0.0;
		Sensor.Alarm.TimeInit := INPUTS.sLocal;
		Sensor.Alarm.AlInit   := TRUE;

		Sensor.AdverVal     := Sensor.Bar;
	ELSE
		Sensor.Alarm.AlLen  := Sensor.Alarm.AlLen + MAIN.Cycle_Time;
	END_IF

	Sensor.Alarm.Alarm := TRUE;
	Sensor.Alarm.Adver := TRUE;

	Sensor.AlErr    := FALSE;
	Sensor.AlMax    := FALSE;
	Sensor.AlMin    := TRUE;
	Sensor.AdverVal := MIN( Sensor.Bar, Sensor.AdverVal );

	Sensor.Alarm.Text     := CONCAT( Sensor.Desc      , ' Underpressured: ' );
	Sensor.Alarm.Text     := CONCAT( Sensor.Alarm.Text, REAL_TO_STRING(Sensor.AdverVal) );

ELSE
	IF Sensor.Alarm.Alarm THEN
		Sensor.Alarm.TimeEnd := INPUTS.sLocal;
		Sensor.Alarm.AlEnd   := TRUE;

	END_IF

	Sensor.Alarm.Alarm := FALSE;
	Sensor.AlErr       := FALSE;
	Sensor.AlMax       := FALSE;
	Sensor.AlMin       := FALSE;

END_IF
END_FUNCTION

(* POU FUN/F_CALC_SENSOR_TEMP, ST *)
FUNCTION F_CALC_SENSOR_TEMP : BOOL
VAR_INPUT
	IN    : REAL;
	Clear : BOOL;
	Cycle : REAL;
END_VAR
VAR_IN_OUT
	Sensor : ST_SENSOR_TEMP;
END_VAR
VAR
END_VAR
(*AVG*)
IF Sensor.Avg_Pos > 4 THEN Sensor.Avg_Pos := 0; END_IF

Sensor.Avg_Sum := Sensor.Avg_Sum + IN - Sensor.Avg_Buf[Sensor.Avg_Pos];
Sensor.Avg_Buf[Sensor.Avg_Pos] := IN;
Sensor.Avg_Pos := Sensor.Avg_Pos + 1;

Sensor.Raw := Sensor.Avg_Sum / 5.0;
Sensor.Err := Sensor.Raw < Sensor.MinRaw OR Sensor.Raw > Sensor.MaxRaw;

(*CALIB*)
Sensor.Deg := Sensor.Raw * Sensor.Cal_K + Sensor.Cal_Off;

(*ALARM*)
IF Clear THEN
	Sensor.Alarm.Alarm := FALSE;
	Sensor.Alarm.Adver := FALSE;
	Sensor.Alarm.AlCnt := 0;
	Sensor.Alarm.AlLen := 0.0;
	Sensor.AdverLv     := 0;
(*	Sensor.AdverVal    := Sensor.Deg;*)

END_IF

IF Sensor.Err THEN
	IF NOT Sensor.Alarm.Alarm THEN
		Sensor.Alarm.AlCnt  := Sensor.Alarm.AlCnt + 1;
		Sensor.Alarm.AlLen  := 0.0;
		Sensor.Alarm.TimeInit := INPUTS.sLocal;
		Sensor.Alarm.AlInit   := TRUE;

		Sensor.Alarm.Text := CONCAT( Sensor.Desc , ' Temperature. Sensor Broken/Disconnected.' );

	ELSE
		Sensor.Alarm.AlLen  := Sensor.Alarm.AlLen + MAIN.Cycle_Time;

	END_IF

	Sensor.Alarm.Alarm := TRUE;
	Sensor.Alarm.Adver := TRUE;

	Sensor.AlErr    := TRUE;
	Sensor.AlLow    := FALSE;
	Sensor.AlHig    := FALSE;
	Sensor.AlMax    := FALSE;
	Sensor.AdverLv  := 4;
	Sensor.AdverVal := 0.0;

ELSIF Sensor.Deg > Sensor.MaxDeg THEN
	IF NOT Sensor.Alarm.Alarm THEN
		Sensor.Alarm.AlCnt  := Sensor.Alarm.AlCnt + 1;
		Sensor.Alarm.AlLen  := 0.0;
		Sensor.Alarm.TimeInit := INPUTS.sLocal;
		Sensor.Alarm.AlInit   := TRUE;

		Sensor.AdverVal     := Sensor.Deg;

	ELSE
		Sensor.Alarm.AlLen  := Sensor.Alarm.AlLen + MAIN.Cycle_Time;

	END_IF

	Sensor.Alarm.Alarm := TRUE;
	Sensor.AlErr       := FALSE;
	Sensor.AlLow       := FALSE;

	IF Sensor.Count > Sensor.Delay THEN
		Sensor.AlHig := FALSE;
		Sensor.AlMax := TRUE;
	ELSE
		Sensor.AlHig := TRUE;
		Sensor.AlMax := FALSE;

		Sensor.Count := Sensor.Count + Cycle;
	END_IF

	IF Sensor.AdverLv < 4 THEN
		Sensor.Alarm.Adver := TRUE;
		Sensor.AdverLv     := 3;
		Sensor.AdverVal    := MAX( Sensor.Deg, Sensor.AdverVal );

		Sensor.Alarm.Text  := CONCAT( Sensor.Desc      , ' Max. Temperature exceeded: '  );
		Sensor.Alarm.Text  := CONCAT( Sensor.Alarm.Text, REAL_TO_STRING(Sensor.AdverVal) );
	END_IF

ELSIF Sensor.Deg > Sensor.HigDeg THEN
	IF NOT Sensor.Alarm.Alarm THEN
		Sensor.Alarm.AlCnt  := Sensor.Alarm.AlCnt + 1;
		Sensor.Alarm.AlLen  := 0.0;
		Sensor.Alarm.TimeInit := INPUTS.sLocal;
		Sensor.Alarm.AlInit   := TRUE;

		Sensor.AdverVal     := Sensor.Deg;

	ELSE
		Sensor.Alarm.AlLen  := Sensor.Alarm.AlLen + MAIN.Cycle_Time;

	END_IF

	Sensor.Alarm.Alarm := TRUE;
	Sensor.AlErr       := FALSE;
	Sensor.AlLow       := FALSE;
	Sensor.AlHig       := TRUE;
	Sensor.AlMax       := FALSE;

	IF Sensor.AdverLv < 3 THEN
		Sensor.Alarm.Adver := TRUE;
		Sensor.AdverLv     := 2;
		Sensor.AdverVal    := MAX( Sensor.Deg, Sensor.AdverVal );

		Sensor.Alarm.Text  := CONCAT( Sensor.Desc      , ' High Temperature exceeded: '  );
		Sensor.Alarm.Text  := CONCAT( Sensor.Alarm.Text, REAL_TO_STRING(Sensor.AdverVal) );
	END_IF

ELSIF Sensor.Deg > Sensor.LowDeg THEN
	Sensor.Alarm.Alarm := FALSE;
	Sensor.AlErr       := FALSE;
	Sensor.AlLow       := TRUE;
	Sensor.AlHig       := FALSE;
	Sensor.AlMax       := FALSE;

	IF Sensor.AdverLv < 2 THEN
		Sensor.Alarm.Adver := TRUE;
		Sensor.AdverLv     := 1;
		Sensor.AdverVal    := MAX( Sensor.Deg, Sensor.AdverVal );

		Sensor.Alarm.Text  := CONCAT( Sensor.Desc      , ' Mild Temperature exceeded: ' );
		Sensor.Alarm.Text  := CONCAT( Sensor.Alarm.Text, REAL_TO_STRING(Sensor.AdverVal) );
	END_IF
ELSE
	IF Sensor.Alarm.Alarm THEN
		Sensor.Alarm.TimeEnd := INPUTS.sLocal;
		Sensor.Alarm.AlEnd   := TRUE;

	END_IF

	Sensor.Alarm.Alarm := FALSE;
	Sensor.AlErr       := FALSE;
	Sensor.AlLow       := FALSE;
	Sensor.AlHig       := FALSE;
	Sensor.AlMax       := FALSE;
	Sensor.Count       := 0;

END_IF
END_FUNCTION

(* POU FUN/F_CALC_SENSOR_POS, ST *)
FUNCTION F_CALC_SENSOR_POS : BOOL
VAR_INPUT
	IN    : REAL;
	Clear : BOOL;
END_VAR
VAR_IN_OUT
	Sensor : ST_SENSOR_POS;
END_VAR
VAR
END_VAR
(*AVG*)
IF Sensor.Avg_Pos > 4 THEN Sensor.Avg_Pos := 0; END_IF

Sensor.Avg_Sum := Sensor.Avg_Sum + IN - Sensor.Avg_Buf[Sensor.Avg_Pos];
Sensor.Avg_Buf[Sensor.Avg_Pos] := IN;
Sensor.Avg_Pos := Sensor.Avg_Pos + 1;

Sensor.Raw := Sensor.Avg_Sum / 5.0;
Sensor.Err := Sensor.Raw < Sensor.MinRaw OR Sensor.Raw > Sensor.MaxRaw;

(*CALIB*)
IF Sensor.Cal_Apply THEN
	IF Sensor.Cal_Min > 0.0 AND Sensor.Cal_Max > 0.0 AND Sensor.Cal_Min <> Sensor.Cal_Max THEN
		Sensor.Cal_K   := 100.0 / (Sensor.Cal_Max - Sensor.Cal_Min);
		Sensor.Cal_Off := -Sensor.Cal_Min * Sensor.Cal_K;

		Sensor.Cal_Min := 0.0;
		Sensor.Cal_Max := 0.0;
	END_IF

	Sensor.Cal_Apply := FALSE;
END_IF

Sensor.Pos := Sensor.Raw * Sensor.Cal_K + Sensor.Cal_Off;

(*ALARM*)
IF Clear THEN
	Sensor.Alarm.Alarm := FALSE;
	Sensor.Alarm.Adver := FALSE;
	Sensor.Alarm.AlCnt := 0;
	Sensor.Alarm.AlLen := 0.0;

END_IF

IF Sensor.Err THEN
	IF NOT Sensor.Alarm.Alarm THEN
		Sensor.Alarm.AlCnt  := Sensor.Alarm.AlCnt + 1;
		Sensor.Alarm.AlLen  := 0.0;
		Sensor.Alarm.TimeInit := INPUTS.sLocal;
		Sensor.Alarm.AlInit   := TRUE;

		Sensor.Alarm.Text   := CONCAT( Sensor.Desc, ' Position. Sensor Broken/Disconnected.' );

	ELSE
		Sensor.Alarm.AlLen  := Sensor.Alarm.AlLen + MAIN.Cycle_Time;
	END_IF

	Sensor.Alarm.Alarm := TRUE;
	Sensor.Alarm.Adver := TRUE;

ELSE
	IF Sensor.Alarm.Alarm THEN
		Sensor.Alarm.TimeEnd := INPUTS.sLocal;
		Sensor.Alarm.AlEnd   := TRUE;

	END_IF

	Sensor.Alarm.Alarm := FALSE;
END_IF
END_FUNCTION

(* POU FUN/F_CALC_SENSOR_KG, ST *)
FUNCTION F_CALC_SENSOR_KG : BOOL
VAR_INPUT
	IN  : REAL;
END_VAR
VAR_IN_OUT
	Sensor : ST_SENSOR_KG;
END_VAR
VAR
END_VAR
Sensor.Raw := IN * Sensor.Cal_K;
Sensor.Kg  := Sensor.Raw * (Sensor.Cal_C / 100.0);
END_FUNCTION

(* POU FUN/F_CALC_CAN_STATE, ST *)
FUNCTION F_CALC_CAN_STATE : BOOL
VAR_INPUT
	State : UINT;
	Clear : BOOL;
END_VAR
VAR_IN_OUT
	Node : ST_CAN_NODESTATE;
END_VAR
VAR
END_VAR
IF Clear THEN
	Node.Alarm.Alarm := FALSE;
	Node.Alarm.Adver := FALSE;
	Node.Alarm.AlCnt := 0;
	Node.Alarm.AlLen := 0.0;
END_IF

IF State <> 0 THEN
	IF NOT Node.Alarm.Alarm THEN
		Node.Alarm.AlCnt  := Node.Alarm.AlCnt + 1;
		Node.Alarm.AlLen  := 0.0;
		Node.Alarm.TimeInit := INPUTS.sLocal;
		Node.Alarm.AlInit   := TRUE;

	ELSE
		Node.Alarm.AlLen  := Node.Alarm.AlLen + MAIN.Cycle_Time;

	END_IF

	Node.Alarm.Adver := TRUE;
	Node.Alarm.Alarm := TRUE;

	Node.Alarm.Text  := CONCAT( Node.Desc  , ' error ' );
	Node.Alarm.Text  := CONCAT( Node.Alarm.Text  , UINT_TO_STRING(State) );

ELSE
	IF Node.Alarm.Alarm THEN
		Node.Alarm.TimeEnd := INPUTS.sLocal;
		Node.Alarm.AlEnd   := TRUE;

	END_IF

	Node.Alarm.Alarm := FALSE;
END_IF
END_FUNCTION

(* POU FUN/F_CALC_CAN_NODESTATE, ST *)
FUNCTION F_CALC_CAN_NODESTATE : BOOL
VAR_INPUT
	State : USINT;
	Clear : BOOL;
END_VAR
VAR_IN_OUT
	Node : ST_CAN_NODESTATE;
END_VAR
IF Clear THEN
	Node.Alarm.Alarm := FALSE;
	Node.Alarm.Adver := FALSE;
	Node.Alarm.AlCnt := 0;
	Node.Alarm.AlLen := 0.0;
END_IF

IF State <> 0 AND State <> 23 THEN
	IF NOT Node.Alarm.Alarm THEN
		Node.Alarm.AlCnt  := Node.Alarm.AlCnt + 1;
		Node.Alarm.AlLen  := 0.0;
		Node.Alarm.TimeInit := INPUTS.sLocal;
		Node.Alarm.AlInit   := TRUE;

	ELSE
		Node.Alarm.AlLen  := Node.Alarm.AlLen + MAIN.Cycle_Time;

	END_IF

	Node.Alarm.Adver := TRUE;
	Node.Alarm.Alarm := TRUE;

	Node.Alarm.Text  := CONCAT( Node.Desc  , ' error ' );
	Node.Alarm.Text  := CONCAT( Node.Alarm.Text  , USINT_TO_STRING(State) );

ELSE
	IF Node.Alarm.Alarm THEN
		Node.Alarm.TimeEnd := INPUTS.sLocal;
		Node.Alarm.AlEnd   := TRUE;

	END_IF

	Node.Alarm.Alarm := FALSE;
END_IF
END_FUNCTION

(* POU FB/FB_DE_CYLINDER_POS, ST *)
FUNCTION_BLOCK FB_DE_CYLINDER_POS
VAR_INPUT
	Enable : BOOL;
	Ready  : BOOL;

	IN_CylIn  : ARRAY[1..2] OF BOOL;
	IN_CylOut : ARRAY[1..2] OF BOOL;
	IN_CylMid : ARRAY[1..2] OF BOOL;
END_VAR
VAR_IN_OUT
	P_In  : ST_SENSOR_BAR;
	P_Out : ST_SENSOR_BAR;
	LS    : ST_SENSOR_POS;
	CFG   : ST_DE_CYLINDER_POS_CFG;
END_VAR
VAR_OUTPUT
	OUT_EV1 : BOOL;
	OUT_EV2 : BOOL;
	OUT_EV3 : BOOL;
	OUT_EV4 : BOOL;

	OUT_HP   : BYTE;
END_VAR
VAR
	State   : WORD;

	IN_Hmi_CylIn  : BOOL;
	IN_Hmi_CylOut : BOOL;
	IN_Hmi_CylMid : BOOL;

	SIIn  : ARRAY[1..3] OF FB_SMART_INPUT;
	SIOut : ARRAY[1..3] OF FB_SMART_INPUT;
	SIMid : ARRAY[1..3] OF FB_SMART_INPUT;

	EventIn  : EN_SMART_INPUT_STATE;
	EventOut : EN_SMART_INPUT_STATE;
	EventMid : EN_SMART_INPUT_STATE;

	TimeCnt : REAL;
	TimeOut : BOOL;

	LS_In  : BOOL;
	LS_Out : BOOL;
	LS_Mid : BOOL;

	ToFaroValue : REAL;
END_VAR
LS_In  := LS.Pos < CFG.TgtLS_In;
LS_Out := LS.Pos > CFG.TgtLS_Out;
LS_Mid := CFG.TgtLS_DB > ABS(CFG.TgtLS_Mid-LS.Pos);

(*Check Inputs*)
SIIn[1](In:= IN_CylIn[1],  T_Cont:= T#0ms, T_DClk:= T#0ms);
SIIn[2](In:= IN_CylIn[2],  T_Cont:= T#0ms, T_DClk:= T#0ms);
SIIn[3](In:= IN_Hmi_CylIn, T_Cont:= T#0ms, T_DClk:= T#0ms);

SIOut[1](In:= IN_CylOut[1],  T_Cont:= T#0ms, T_DClk:= T#0ms);
SIOut[2](In:= IN_CylOut[2],  T_Cont:= T#0ms, T_DClk:= T#0ms);
SIOut[3](In:= IN_Hmi_CylOut, T_Cont:= T#0ms, T_DClk:= T#0ms);

SIMid[1](In:= IN_CylMid[1],  T_Cont:= T#0ms, T_DClk:= T#0ms);
SIMid[2](In:= IN_CylMid[2],  T_Cont:= T#0ms, T_DClk:= T#0ms);
SIMid[3](In:= IN_Hmi_CylMid, T_Cont:= T#0ms, T_DClk:= T#0ms);

IF NOT Enable THEN
	OUT_EV1 := FALSE;
	OUT_EV2 := FALSE;
	OUT_EV3 := FALSE;
	OUT_EV4 := FALSE;

	OUT_HP  := 0;

	ToFaroValue := 0.0;

	TimeCnt := 0.0;
	State   := 0;
	RETURN;
END_IF

(*Check Time*)
TimeOut := TimeOut OR ( CFG.TimeMax > 0  AND TimeCnt > CFG.TimeMax );
TimeCnt := TimeCnt + CFG.Cycle;

IF    SIIn[1].Event <> NONE THEN EventIn := SIIn[1].Event;
ELSIF SIIn[2].Event <> NONE THEN EventIn := SIIn[2].Event;
ELSIF SIIn[3].Event <> NONE THEN EventIn := SIIn[3].Event;
ELSE
	EventIn := NONE;
END_IF

IF    SIOut[1].Event <> NONE THEN EventOut := SIOut[1].Event;
ELSIF SIOut[2].Event <> NONE THEN EventOut := SIOut[2].Event;
ELSIF SIOut[3].Event <> NONE THEN EventOut := SIOut[3].Event;
ELSE
	EventOut := NONE;
END_IF

IF    SIMid[1].Event <> NONE THEN EventMid := SIMid[1].Event;
ELSIF SIMid[2].Event <> NONE THEN EventMid := SIMid[2].Event;
ELSIF SIMid[3].Event <> NONE THEN EventMid := SIMid[3].Event;
ELSE
	EventMid := NONE;
END_IF

(*Working States*)
CASE State OF

(*Init State*)
0:
	ToFaroValue := 0.0;

	(*Start Manual IN*)
	IF EventIn = INIT_CONTINUOUS AND Ready AND NOT P_In.AlMax AND NOT (CFG.LS_Limit_In AND (LS_In OR LS.Err)) THEN
		OUT_EV1  := FALSE;
		OUT_EV2  := TRUE;
		OUT_EV3  := TRUE;
		OUT_EV4  := FALSE;
		OUT_HP   := CFG.HP;

		TimeOut := FALSE; (*Reset TimeOut Error*)
		State   := 1100;  (*Next State*)

		ToFaroValue := 1.0;

	(*Start Manual OUT*)
	ELSIF EventOut = INIT_CONTINUOUS AND Ready AND NOT P_Out.AlMax AND NOT (CFG.LS_Limit_Out AND (LS_Out OR LS.Err)) THEN
		OUT_EV1  := TRUE;
		OUT_EV2  := FALSE;
		OUT_EV3  := FALSE;
		OUT_EV4  := TRUE;
		OUT_HP   := CFG.HP;

		TimeOut := FALSE; (*Reset TimeOut Error*)
		State   := 2100;  (*Next State*)

		ToFaroValue := -1.0;

	(*Start Manual MID*)
	ELSIF EventMid = INIT_CONTINUOUS AND Ready AND NOT LS_Mid AND NOT LS.Err THEN
		IF LS.Pos > CFG.TgtLS_Mid AND NOT P_In.AlMax THEN
			OUT_EV1  := FALSE;
			OUT_EV2  := TRUE;
			OUT_EV3  := TRUE;
			OUT_EV4  := FALSE;
			OUT_HP   := CFG.HP;

			TimeOut := FALSE; (*Reset TimeOut Error*)
			State   := 1200;  (*Next State*)

			ToFaroValue := 1.0;

		ELSIF NOT P_Out.AlMax THEN
			OUT_EV1  := TRUE;
			OUT_EV2  := FALSE;
			OUT_EV3  := FALSE;
			OUT_EV4  := TRUE;
			OUT_HP   := CFG.HP;

			TimeOut := FALSE; (*Reset TimeOut Error*)
			State   := 2200;  (*Next State*)

			ToFaroValue := -1.0;

		END_IF

	(*Nothing*)
	ELSE
		OUT_EV1  := FALSE;
		OUT_EV2  := FALSE;
		OUT_EV3  := FALSE;
		OUT_EV4  := FALSE;
		OUT_HP   := 0;

	END_IF

    TimeCnt := 0.0; (*Time Count*)

(*Manual IN*)
1100:
	(*End IN*)
	IF EventIn <> NONE OR EventOut <> NONE OR TimeOut OR P_In.AlMax OR CFG.LS_Limit_In AND (LS_In OR LS.Err) THEN
		OUT_EV1  := FALSE;
		OUT_EV2  := FALSE;
		OUT_EV3  := FALSE;
		OUT_EV4  := FALSE;
		OUT_HP   := 0;

		State := 0; (*Next State*)

	END_IF

(*Manual MID*)
1200:
	(*End IN*)
	IF EventIn <> NONE OR EventOut <> NONE OR TimeOut OR P_In.AlMax OR LS_Mid THEN
		OUT_EV1  := FALSE;
		OUT_EV2  := FALSE;
		OUT_EV3  := FALSE;
		OUT_EV4  := FALSE;
		OUT_HP   := 0;

		State := 0; (*Next State*)

	END_IF

(*Manual OUT*)
2100:
	(*End OUT*)
	IF EventOut <> NONE OR EventIn <> NONE OR TimeOut OR P_Out.AlMax OR CFG.LS_Limit_Out AND (LS_Out OR LS.Err) THEN
		OUT_EV1  := FALSE;
		OUT_EV2  := FALSE;
		OUT_EV3  := FALSE;
		OUT_EV4  := FALSE;
		OUT_HP   := CFG.HP;

		State := 0; (*Next State*)

	END_IF

(*Manual OUT*)
2200:
	(*End OUT*)
	IF EventOut <> NONE OR EventIn <> NONE OR TimeOut OR P_Out.AlMax OR LS_Mid THEN
		OUT_EV1  := FALSE;
		OUT_EV2  := FALSE;
		OUT_EV3  := FALSE;
		OUT_EV4  := FALSE;
		OUT_HP   := CFG.HP;

		State := 0; (*Next State*)

	END_IF

END_CASE
END_FUNCTION_BLOCK

(* POU FB/FB_BACKSTAY, ST *)
FUNCTION_BLOCK FB_BACKSTAY
VAR_INPUT
	Enable : BOOL;
	Ready  : BOOL;

	IN_P_In   : ARRAY[1..2] OF BOOL;
	IN_P_Out  : ARRAY[1..2] OF BOOL;
	IN_S_In   : ARRAY[1..2] OF BOOL;
	IN_S_Out  : ARRAY[1..2] OF BOOL;

END_VAR
VAR_IN_OUT
	P_P  : ST_SENSOR_BAR;
	P_S  : ST_SENSOR_BAR;
	LS_P : ST_SENSOR_POS;
	LS_S : ST_SENSOR_POS;
	CFG  : ST_SE_CYLINDER_POS_CFG;
END_VAR
VAR_OUTPUT
	OUT_P_In  : BOOL;
	OUT_P_Out : BOOL;
	OUT_S_In  : BOOL;
	OUT_S_Out : BOOL;

	OUT_HP    : BYTE;
END_VAR
VAR
	State   : WORD;
	State_P : WORD;
	State_S : WORD;

	IN_Hmi_P_In  : BOOL;
	IN_Hmi_P_Out : BOOL;
	IN_Hmi_S_In  : BOOL;
	IN_Hmi_S_Out : BOOL;

	SI_P_In  : ARRAY[1..3] OF FB_SMART_INPUT;
	SI_P_Out : ARRAY[1..3] OF FB_SMART_INPUT;
	SI_S_In  : ARRAY[1..3] OF FB_SMART_INPUT;
	SI_S_Out : ARRAY[1..3] OF FB_SMART_INPUT;

	Event_P_In  : EN_SMART_INPUT_STATE;
	Event_P_Out : EN_SMART_INPUT_STATE;
	Event_S_In  : EN_SMART_INPUT_STATE;
	Event_S_Out : EN_SMART_INPUT_STATE;

	TimeCnt : REAL;
	TimeOut : BOOL;

	Slow_P : BOOL;
	Slow_S : BOOL;

	LS_P_In  : BOOL;
	LS_P_Out : BOOL;
	LS_S_In  : BOOL;
	LS_S_Out : BOOL;

	ToFaroValueP : REAL;
	ToFaroValueS : REAL;

END_VAR
LS_P_Out := LS_P.Pos > CFG.TgtLS_Out;
LS_P_In  := LS_P.Pos < CFG.TgtLS_In;
LS_S_Out := LS_S.Pos > CFG.TgtLS_Out;
LS_S_In  := LS_S.Pos < CFG.TgtLS_In;

(*Check Inputs*)
SI_P_In[1](In:= IN_P_In[1],  T_Cont:= T#0ms, T_DClk:= T#0ms);
SI_P_In[2](In:= IN_P_In[2],  T_Cont:= T#0ms, T_DClk:= T#0ms);
SI_P_In[3](In:= IN_Hmi_P_In, T_Cont:= T#0ms, T_DClk:= T#0ms);

SI_P_Out[1](In:= IN_P_Out[1],  T_Cont:= T#0ms, T_DClk:= T#0ms);
SI_P_Out[2](In:= IN_P_Out[2],  T_Cont:= T#0ms, T_DClk:= T#0ms);
SI_P_Out[3](In:= IN_Hmi_P_Out, T_Cont:= T#0ms, T_DClk:= T#0ms);

SI_S_In[1](In:= IN_S_In[1],  T_Cont:= T#0ms, T_DClk:= T#0ms);
SI_S_In[2](In:= IN_S_In[2],  T_Cont:= T#0ms, T_DClk:= T#0ms);
SI_S_In[3](In:= IN_Hmi_S_In, T_Cont:= T#0ms, T_DClk:= T#0ms);

SI_S_Out[1](In:= IN_S_Out[1],  T_Cont:= T#0ms, T_DClk:= T#0ms);
SI_S_Out[2](In:= IN_S_Out[2],  T_Cont:= T#0ms, T_DClk:= T#0ms);
SI_S_Out[3](In:= IN_Hmi_S_Out, T_Cont:= T#0ms, T_DClk:= T#0ms);

IF NOT Enable THEN
	OUT_P_In  := FALSE;
	OUT_P_Out := FALSE;
	OUT_S_In  := FALSE;
	OUT_S_Out := FALSE;
	OUT_HP    := 0;

	ToFaroValueP := 0.0;
	ToFaroValueS := 0.0;

	TimeCnt := 0.0;
	State   := 0;
	State_P := 0;
	State_S := 0;
	RETURN;
END_IF

(*Check Time*)
TimeOut := TimeOut OR ( CFG.TimeMax > 0  AND TimeCnt > CFG.TimeMax );
TimeCnt := TimeCnt + CFG.Cycle;

IF    SI_P_In[1].Event <> NONE THEN Event_P_In := SI_P_In[1].Event; Slow_P := FALSE;
ELSIF SI_P_In[2].Event <> NONE THEN Event_P_In := SI_P_In[2].Event; Slow_P := TRUE;
ELSIF SI_P_In[3].Event <> NONE THEN Event_P_In := SI_P_In[3].Event; Slow_P := TRUE;
ELSE
	Event_P_In := NONE;
END_IF

IF    SI_P_Out[1].Event <> NONE THEN Event_P_Out := SI_P_Out[1].Event;
ELSIF SI_P_Out[2].Event <> NONE THEN Event_P_Out := SI_P_Out[2].Event;
ELSIF SI_P_Out[3].Event <> NONE THEN Event_P_Out := SI_P_Out[3].Event;
ELSE
	Event_P_Out := NONE;
END_IF

IF    SI_S_In[1].Event <> NONE THEN Event_S_In := SI_S_In[1].Event; Slow_S := FALSE;
ELSIF SI_S_In[2].Event <> NONE THEN Event_S_In := SI_S_In[2].Event; Slow_S := TRUE;
ELSIF SI_S_In[3].Event <> NONE THEN Event_S_In := SI_S_In[3].Event; Slow_S := TRUE;
ELSE
	Event_S_In := NONE;
END_IF

IF    SI_S_Out[1].Event <> NONE THEN Event_S_Out := SI_S_Out[1].Event;
ELSIF SI_S_Out[2].Event <> NONE THEN Event_S_Out := SI_S_Out[2].Event;
ELSIF SI_S_Out[3].Event <> NONE THEN Event_S_Out := SI_S_Out[3].Event;
ELSE
	Event_S_Out := NONE;
END_IF


(*Common Working States*)
CASE State OF

(*Common Init State*)
0:

	OUT_HP := 0;

	IF State_P = 0 AND State_S = 0 THEN TimeCnt := 0.0; END_IF

(*Port Working States*)
	CASE State_P OF
	(*Init State*)
	0:
		ToFaroValueP := 0.0;

		(*Start Manual IN*)
		IF Event_P_In = INIT_CONTINUOUS AND Ready AND NOT P_P.AlMax AND NOT (CFG.LS_Limit_In AND (LS_P_In OR LS_P.Err)) THEN
			OUT_P_In  := TRUE;
			OUT_P_Out := FALSE;

			TimeOut   := FALSE; (*Reset TimeOut Error*)
			State_P   := 1100;  (*Next State*)

			ToFaroValueP := 1.0;
	
		(*Start Manual OUT*)
		ELSIF Event_P_Out = INIT_CONTINUOUS AND NOT (CFG.LS_Limit_Out AND (LS_P_Out OR LS_P.Err)) THEN
			OUT_P_In  := FALSE;
			OUT_P_Out := TRUE;

			TimeOut   := FALSE; (*Reset TimeOut Error*)
			State_P   := 2100;  (*Next State*)

			ToFaroValueP := -1.0;

		(*Nothing*)
		ELSE
			OUT_P_In  := FALSE;
			OUT_P_Out := FALSE;

		END_IF

	(*Manual IN*)
	1100:
		(*End IN*)
		IF Event_P_In <> NONE OR Event_P_Out <> NONE OR TimeOut OR P_P.AlMax OR CFG.LS_Limit_In AND (LS_P_In OR LS_P.Err) THEN
			OUT_P_In  := FALSE;
			OUT_P_Out := FALSE;

			State_P   := 0; (*Next State*)

		ELSIF Slow_P OR Slow_S THEN
			OUT_HP := 1;

		ELSE
			OUT_HP := CFG.HP;

		END_IF

	(*Manual OUT*)
	2100:
		(*End OUT*)
		IF Event_P_Out <> NONE OR Event_P_In <> NONE OR TimeOut OR CFG.LS_Limit_Out AND (LS_P_Out OR LS_P.Err)THEN
			OUT_P_In  := FALSE;
			OUT_P_Out := FALSE;

			State_P   := 0; (*Next State*)
		END_IF

	END_CASE

(*Stbd Working States*)
	CASE State_S OF
	(*Init State*)
	0:
		ToFaroValueS := 0.0;

		(*Start Manual IN*)
		IF Event_S_In = INIT_CONTINUOUS AND Ready AND NOT P_S.AlMax AND NOT (CFG.LS_Limit_In AND (LS_S_In OR LS_S.Err)) THEN
			OUT_S_In  := TRUE;
			OUT_S_Out := FALSE;

			TimeOut   := FALSE; (*Reset TimeOut Error*)
			State_S   := 1100;  (*Next State*)

			ToFaroValueS := 1.0;

		(*Start Manual OUT*)
		ELSIF Event_S_Out = INIT_CONTINUOUS AND NOT (CFG.LS_Limit_Out AND (LS_S_Out OR LS_S.Err)) THEN
			OUT_S_In  := FALSE;
			OUT_S_Out := TRUE;

			TimeOut   := FALSE; (*Reset TimeOut Error*)
			State_S   := 2100;  (*Next State*)

			ToFaroValueS := -1.0;

		(*Nothing*)
		ELSE
			OUT_S_In  := FALSE;
			OUT_S_Out := FALSE;

		END_IF

	(*Manual IN*)
	1100:
		(*End IN*)
		IF Event_S_In <> NONE OR Event_S_Out <> NONE OR TimeOut OR P_S.AlMax OR CFG.LS_Limit_In AND (LS_S_In OR LS_S.Err) THEN
			OUT_S_In  := FALSE;
			OUT_S_Out := FALSE;

			State_S   := 0; (*Next State*)

		ELSIF Slow_P OR Slow_S THEN
			OUT_HP := 1;

		ELSE
			OUT_HP := CFG.HP;

		END_IF

	(*Manual OUT*)
	2100:
		(*End OUT*)
		IF Event_S_Out <> NONE OR Event_S_In <> NONE OR TimeOut OR CFG.LS_Limit_Out AND (LS_S_Out OR LS_S.Err)THEN
			OUT_S_In  := FALSE;
			OUT_S_Out := FALSE;

			State_S   := 0; (*Next State*)
		END_IF

	END_CASE

END_CASE
END_FUNCTION_BLOCK

(* POU FB/FB_WATERBALLAST, ST *)
FUNCTION_BLOCK FB_WATERBALLAST
VAR_INPUT
	Enable : BOOL;
	Ready  : BOOL;

	Perc : REAL;

	IN_P_Fwd : ARRAY[1..2] OF BOOL;
	IN_P_Aft : ARRAY[1..2] OF BOOL;
	IN_S_Fwd : ARRAY[1..2] OF BOOL;
	IN_S_Aft : ARRAY[1..2] OF BOOL;
	IN_Fill  : ARRAY[1..2] OF BOOL;
	IN_12    : ARRAY[1..2] OF BOOL;
	IN_Dump  : ARRAY[1..2] OF BOOL;
	IN_Move  : ARRAY[1..2] OF BOOL;
	IN_Stop  : ARRAY[1..2] OF BOOL;

	SF_P_Fwd : BOOL;
	SF_P_Aft : BOOL;
	SF_S_Fwd : BOOL;
	SF_S_Aft : BOOL;
END_VAR
VAR_IN_OUT

	WB_A : FB_WB_VALVE;
	WB_B : FB_WB_VALVE_LS;
	WB_C : FB_WB_VALVE_LS;
	WB_D : FB_WB_VALVE;
	WB_E : FB_WB_VALVE;
	WB_F : FB_WB_VALVE;
	WB_G : FB_WB_VALVE;
	WB_H : FB_WB_VALVE;
	WB_I : FB_WB_VALVE_LS;
	WB_J : FB_WB_VALVE;
	WB_K : FB_WB_VALVE;
	WB_L : FB_WB_VALVE;
	WB_M : FB_WB_VALVE;
	WB_N : FB_WB_VALVE_LS;
	WB_R : FB_WB_VALVE_LS;
	WB_S : FB_WB_VALVE_LS;

	WB_PUD : FB_WB_VALVE_LS;
    WB_PAF : FB_WB_VALVE_LS;
	WB_SUD : FB_WB_VALVE_LS;
    WB_SAF : FB_WB_VALVE_LS;

	CFG : ST_WB_CFG;
END_VAR
VAR_OUTPUT
	EVP_Pump : INT; (*%*)
	OUT_LP   : BYTE;

	OUT_P_Fwd : BOOL;
	OUT_P_Aft : BOOL;
	OUT_S_Fwd : BOOL;
	OUT_S_Aft : BOOL;
	OUT_Fill  : BOOL;
	OUT_12    : BOOL;
	OUT_Dump  : BOOL;
	OUT_Move  : BOOL;
	OUT_Stop  : BOOL;
	OUT_Pump  : BOOL;
END_VAR
VAR
	State : WORD;
	Next  : WORD;
	Error : WORD;

	IN_Hmi_P_Fwd : BOOL;
	IN_Hmi_P_Aft : BOOL;
	IN_Hmi_S_Fwd : BOOL;
	IN_Hmi_S_Aft : BOOL;
	IN_Hmi_Fill  : BOOL;
	IN_Hmi_12    : BOOL;
	IN_Hmi_Dump  : BOOL;
	IN_Hmi_Move  : BOOL;
	IN_Hmi_Stop  : BOOL;

	IN_Hmi_Pump  : BOOL;
	IN_Hmi_Pump_Perc  : INT := 20;


	SI_P_Fwd : ARRAY[1..3] OF FB_SMART_INPUT;
	SI_P_Aft : ARRAY[1..3] OF FB_SMART_INPUT;
	SI_S_Fwd : ARRAY[1..3] OF FB_SMART_INPUT;
	SI_S_Aft : ARRAY[1..3] OF FB_SMART_INPUT;
	SI_Fill  : ARRAY[1..3] OF FB_SMART_INPUT;
	SI_12    : ARRAY[1..3] OF FB_SMART_INPUT;
	SI_Dump  : ARRAY[1..3] OF FB_SMART_INPUT;
	SI_Move  : ARRAY[1..3] OF FB_SMART_INPUT;
	SI_Stop  : ARRAY[1..3] OF FB_SMART_INPUT;
	SI_Break : ARRAY[1..3] OF FB_SMART_INPUT;

	SI_Pump : FB_SMART_INPUT;

	Event_P_Fwd : EN_SMART_INPUT_STATE;
	Event_P_Aft : EN_SMART_INPUT_STATE;
	Event_S_Fwd : EN_SMART_INPUT_STATE;
	Event_S_Aft : EN_SMART_INPUT_STATE;
	Event_Fill  : EN_SMART_INPUT_STATE;
	Event_12    : EN_SMART_INPUT_STATE;
	Event_Dump  : EN_SMART_INPUT_STATE;
	Event_Move  : EN_SMART_INPUT_STATE;
	Event_Stop  : EN_SMART_INPUT_STATE;
    Event_Break : EN_SMART_INPUT_STATE;

	NewEvent : BOOL;
	TimeCnt  : REAL;
	TimeDump : REAL;
	TimeMove : REAL;

	EVP_Pump_Tgt  : REAL;
	SoftStop      : BOOL;

	Init          : BOOL;
	Pause         : BOOL;

END_VAR
VAR PERSISTENT
	Manual AT %Q*: BOOL;
END_VAR
(*Check Inputs*)
SI_P_Fwd[1](In:= IN_P_Fwd[1],  T_Cont:= T#0ms, T_DClk:= T#0ms);
SI_P_Fwd[2](In:= IN_P_Fwd[2],  T_Cont:= T#0ms, T_DClk:= T#0ms);
SI_P_Fwd[3](In:= IN_Hmi_P_Fwd, T_Cont:= T#0ms, T_DClk:= T#0ms);

SI_P_Aft[1](In:= IN_P_Aft[1],  T_Cont:= T#0ms, T_DClk:= T#0ms);
SI_P_Aft[2](In:= IN_P_Aft[2],  T_Cont:= T#0ms, T_DClk:= T#0ms);
SI_P_Aft[3](In:= IN_Hmi_P_Aft, T_Cont:= T#0ms, T_DClk:= T#0ms);

SI_S_Fwd[1](In:= IN_S_Fwd[1],  T_Cont:= T#0ms, T_DClk:= T#0ms);
SI_S_Fwd[2](In:= IN_S_Fwd[2],  T_Cont:= T#0ms, T_DClk:= T#0ms);
SI_S_Fwd[3](In:= IN_Hmi_S_Fwd, T_Cont:= T#0ms, T_DClk:= T#0ms);

SI_S_Aft[1](In:= IN_S_Aft[1],  T_Cont:= T#0ms, T_DClk:= T#0ms);
SI_S_Aft[2](In:= IN_S_Aft[2],  T_Cont:= T#0ms, T_DClk:= T#0ms);
SI_S_Aft[3](In:= IN_Hmi_S_Aft, T_Cont:= T#0ms, T_DClk:= T#0ms);

SI_12[1](In:= IN_12[1],  T_Cont:= T#0ms, T_DClk:= T#0ms);
SI_12[2](In:= IN_12[2],  T_Cont:= T#0ms, T_DClk:= T#0ms);
SI_12[3](In:= IN_Hmi_12, T_Cont:= T#0ms, T_DClk:= T#0ms);

SI_Fill[1](In:= IN_Fill[1],  T_Cont:= T#0ms, T_DClk:= T#0ms);
SI_Fill[2](In:= IN_Fill[2],  T_Cont:= T#0ms, T_DClk:= T#0ms);
SI_Fill[3](In:= IN_Hmi_Fill, T_Cont:= T#0ms, T_DClk:= T#0ms);

SI_Dump[1](In:= IN_Dump[1],  T_Cont:= T#0ms, T_DClk:= T#0ms);
SI_Dump[2](In:= IN_Dump[2],  T_Cont:= T#0ms, T_DClk:= T#0ms);
SI_Dump[3](In:= IN_Hmi_Dump, T_Cont:= T#0ms, T_DClk:= T#0ms);

SI_Move[1](In:= IN_Move[1],  T_Cont:= T#0ms, T_DClk:= T#0ms);
SI_Move[2](In:= IN_Move[2],  T_Cont:= T#0ms, T_DClk:= T#0ms);
SI_Move[3](In:= IN_Hmi_Move, T_Cont:= T#0ms, T_DClk:= T#0ms);

SI_Stop[1](In:= IN_Stop[1],  T_Cont:= T#0ms, T_DClk:= T#0ms);
SI_Stop[2](In:= IN_Stop[2],  T_Cont:= T#0ms, T_DClk:= T#0ms);
SI_Stop[3](In:= IN_Hmi_Stop, T_Cont:= T#0ms, T_DClk:= T#0ms);

SI_Break[1](In:= IN_Stop[1],  T_Cont:= T#2000ms, T_DClk:= T#0ms);
SI_Break[2](In:= IN_Stop[2],  T_Cont:= T#2000ms, T_DClk:= T#0ms);
SI_Break[3](In:= IN_Hmi_Stop, T_Cont:= T#2000ms, T_DClk:= T#0ms);

SI_Pump(In:= IN_Hmi_Pump, T_Cont:= T#0ms, T_DClk:= T#0ms);

IF NOT Enable THEN
	EVP_Pump := 0;
	OUT_LP   := 0;

	TimeCnt := 0.0;
	State   := 0;
	RETURN;
END_IF

IF    SI_P_Fwd[1].Event <> NONE THEN Event_P_Fwd := SI_P_Fwd[1].Event;
ELSIF SI_P_Fwd[2].Event <> NONE THEN Event_P_Fwd := SI_P_Fwd[2].Event;
ELSIF SI_P_Fwd[3].Event <> NONE THEN Event_P_Fwd := SI_P_Fwd[3].Event;
ELSE
	Event_P_Fwd := NONE;
END_IF

IF    SI_P_Aft[1].Event <> NONE THEN Event_P_Aft := SI_P_Aft[1].Event;
ELSIF SI_P_Aft[2].Event <> NONE THEN Event_P_Aft := SI_P_Aft[2].Event;
ELSIF SI_P_Aft[3].Event <> NONE THEN Event_P_Aft := SI_P_Aft[3].Event;
ELSE
	Event_P_Aft := NONE;
END_IF

IF    SI_S_Fwd[1].Event <> NONE THEN Event_S_Fwd := SI_S_Fwd[1].Event;
ELSIF SI_S_Fwd[2].Event <> NONE THEN Event_S_Fwd := SI_S_Fwd[2].Event;
ELSIF SI_S_Fwd[3].Event <> NONE THEN Event_S_Fwd := SI_S_Fwd[3].Event;
ELSE
	Event_S_Fwd := NONE;
END_IF

IF    SI_S_Aft[1].Event <> NONE THEN Event_S_Aft := SI_S_Aft[1].Event;
ELSIF SI_S_Aft[2].Event <> NONE THEN Event_S_Aft := SI_S_Aft[2].Event;
ELSIF SI_S_Aft[3].Event <> NONE THEN Event_S_Aft := SI_S_Aft[3].Event;
ELSE
	Event_S_Aft := NONE;
END_IF

IF    SI_Fill[1].Event <> NONE THEN Event_Fill := SI_Fill[1].Event;
ELSIF SI_Fill[2].Event <> NONE THEN Event_Fill := SI_Fill[2].Event;
ELSIF SI_Fill[3].Event <> NONE THEN Event_Fill := SI_Fill[3].Event;
ELSE
	Event_Fill := NONE;
END_IF

IF    SI_12[1].Event <> NONE THEN Event_12 := SI_12[1].Event;
ELSIF SI_12[2].Event <> NONE THEN Event_12 := SI_12[2].Event;
ELSIF SI_12[3].Event <> NONE THEN Event_12 := SI_12[3].Event;
ELSE
	Event_12 := NONE;
END_IF

IF    SI_Dump[1].Event <> NONE THEN Event_Dump := SI_Dump[1].Event;
ELSIF SI_Dump[2].Event <> NONE THEN Event_Dump := SI_Dump[2].Event;
ELSIF SI_Dump[3].Event <> NONE THEN Event_Dump := SI_Dump[3].Event;
ELSE
	Event_Dump := NONE;
END_IF

IF    SI_Move[1].Event <> NONE THEN Event_Move := SI_Move[1].Event;
ELSIF SI_Move[2].Event <> NONE THEN Event_Move := SI_Move[2].Event;
ELSIF SI_Move[3].Event <> NONE THEN Event_Move := SI_Move[3].Event;
ELSE
	Event_Move := NONE;
END_IF

IF    SI_Stop[1].Event <> NONE THEN Event_Stop := SI_Stop[1].Event;
ELSIF SI_Stop[2].Event <> NONE THEN Event_Stop := SI_Stop[2].Event;
ELSIF SI_Stop[3].Event <> NONE THEN Event_Stop := SI_Stop[3].Event;
ELSE
	Event_Stop := NONE;
END_IF

IF    SI_Break[1].Event <> NONE THEN Event_Break := SI_Break[1].Event;
ELSIF SI_Break[2].Event <> NONE THEN Event_Break := SI_Break[2].Event;
ELSIF SI_Break[3].Event <> NONE THEN Event_Break := SI_Break[3].Event;
ELSE
	Event_Break := NONE;
END_IF

(*Check Time*)
(*TimeOut := TimeOut OR ( CFG.TimeMax > 0  AND TimeCnt > CFG.TimeMax );*)
TimeCnt := TimeCnt  + CFG.Cycle;

(*Working States*)
CASE State OF

(*Init State*)
0:
	EVP_Pump_Tgt := CFG.EVP_Pump_Min;
	EVP_Pump := 0;
	OUT_LP   := 0;

    OUT_Fill := FALSE;
    OUT_Dump := FALSE;
    OUT_Move := FALSE;
    OUT_Stop := FALSE;

	Pause    := FALSE;
	SoftStop := FALSE;

	WB_A.B_Close := FALSE;
	WB_B.B_Close := FALSE;
	WB_C.B_Close := FALSE;
	WB_D.B_Close := FALSE;
	WB_E.B_Close := FALSE;
	WB_F.B_Close := FALSE;
	WB_G.B_Close := FALSE;
	WB_H.B_Close := FALSE;
	WB_I.B_Close := FALSE;
	WB_J.B_Close := FALSE;
	WB_K.B_Close := FALSE;
	WB_L.B_Close := FALSE;
	WB_M.B_Close := FALSE;
	WB_N.B_Close := FALSE;
	WB_R.B_Close := FALSE;
	WB_S.B_Close := FALSE;

	WB_PUD.B_Close := FALSE;
	WB_PAF.B_Close := FALSE;
	WB_SUD.B_Close := FALSE;
	WB_SAF.B_Close := FALSE;

	WB_A.B_Open := FALSE;
	WB_B.B_Open := FALSE;
	WB_C.B_Open := FALSE;
	WB_D.B_Open := FALSE;
	WB_E.B_Open := FALSE;
	WB_F.B_Open := FALSE;
	WB_G.B_Open := FALSE;
	WB_H.B_Open := FALSE;
	WB_I.B_Open := FALSE;
	WB_J.B_Open := FALSE;
	WB_K.B_Open := FALSE;
	WB_L.B_Open := FALSE;
	WB_M.B_Open := FALSE;
	WB_N.B_Open := FALSE;
	WB_R.B_Open := FALSE;
	WB_S.B_Open := FALSE;

	WB_PUD.B_Open := FALSE;
	WB_PAF.B_Open := FALSE;
	WB_SUD.B_Open := FALSE;
	WB_SAF.B_Open := FALSE;

	WB_PUD.B_Half := FALSE;
	WB_SUD.B_Half := FALSE;

	(*Manual*)
	IF Manual THEN
		OUT_P_Fwd := FALSE;
		OUT_P_Aft := FALSE;
		OUT_S_Fwd := FALSE;
		OUT_S_Aft := FALSE;
		OUT_12    := FALSE;
		TimeCnt   := 0.0;

		IF SI_Pump.Event = INIT_CONTINUOUS AND Ready THEN
			EVP_Pump_Tgt := CFG.EVP_Pump_Min;

			EVP_Pump := REAL_TO_INT(EVP_Pump_Tgt * Perc * 10.0);
			OUT_LP   := 1;
			State    := 100;   (*Next State*)

		END_IF

	(*Automatico*)
	ELSE
		IF Event_P_Fwd = INIT_CONTINUOUS THEN
			OUT_P_Fwd := TRUE;
			OUT_P_Aft := FALSE;
			OUT_S_Fwd := FALSE;
			OUT_S_Aft := FALSE;
			TimeCnt   := 0.0;
		ELSIF Event_P_Aft = INIT_CONTINUOUS THEN
			OUT_P_Fwd := FALSE;
			OUT_P_Aft := TRUE;
			OUT_S_Fwd := FALSE;
			OUT_S_Aft := FALSE;
			TimeCnt   := 0.0;
		ELSIF Event_S_Fwd = INIT_CONTINUOUS THEN
			OUT_P_Fwd := FALSE;
			OUT_P_Aft := FALSE;
			OUT_S_Fwd := TRUE;
			OUT_S_Aft := FALSE;
			TimeCnt   := 0.0;
		ELSIF Event_S_Aft = INIT_CONTINUOUS THEN
			OUT_P_Fwd := FALSE;
			OUT_P_Aft := FALSE;
			OUT_S_Fwd := FALSE;
			OUT_S_Aft := TRUE;
			TimeCnt   := 0.0;
		END_IF

		IF Event_12 = INIT_CONTINUOUS THEN
			OUT_12  := NOT OUT_12;
			TimeCnt := 0.0;
		END_IF

		IF Event_Stop = INIT_CONTINUOUS OR TimeCnt > CFG.TimeMax_Idle THEN
			OUT_P_Fwd := FALSE;
			OUT_P_Aft := FALSE;
			OUT_S_Fwd := FALSE;
			OUT_S_Aft := FALSE;
			OUT_12    := FALSE;
		END_IF

		IF Event_Fill = INIT_CONTINUOUS THEN

			IF    Out_P_Fwd THEN State := 5000; Next := 1010;
			ELSIF Out_P_Aft THEN State := 5000; Next := 1020;
			ELSIF Out_S_Fwd THEN State := 5000; Next := 1030;
			ELSIF Out_S_Aft THEN State := 5000; Next := 1040;
			END_IF

			OUT_Fill := TRUE;
			Error    := 0;
			TimeCnt  := 0.0;

		ELSIF Event_Dump = INIT_CONTINUOUS THEN

			IF    Out_P_Fwd THEN State := 5000; Next := 2010; TimeDump := CFG.TimeMax_DumpFwd;
			ELSIF Out_P_Aft THEN State := 5000; Next := 2020; TimeDump := CFG.TimeMax_DumpAft;
			ELSIF Out_S_Fwd THEN State := 5000; Next := 2030; TimeDump := CFG.TimeMax_DumpFwd;
			ELSIF Out_S_Aft THEN State := 5000; Next := 2040; TimeDump := CFG.TimeMax_DumpAft;
			END_IF

			OUT_Dump := TRUE;
			Error    := 0;
			TimeCnt  := 0.0;

		ELSIF Event_Move = INIT_CONTINUOUS THEN

			IF    Out_P_Fwd THEN State := 5000; Next := 3010; TimeMove := CFG.TimeMax_MoveFwd;
			ELSIF Out_P_Aft THEN State := 5000; Next := 3020; TimeMove := CFG.TimeMax_MoveAft;
			ELSIF Out_S_Fwd THEN State := 5000; Next := 3030; TimeMove := CFG.TimeMax_MoveFwd;
			ELSIF Out_S_Aft THEN State := 5000; Next := 3040; TimeMove := CFG.TimeMax_MoveAft;
			END_IF

			OUT_Move := TRUE;
			Error    := 0;
			TimeCnt  := 0.0;

		ELSIF Event_Break = INIT_CONTINUOUS THEN

			Error    := 0;
			TimeCnt  := 0.0;
			State    := 5000;
			Next     := 0;

		END_IF

	END_IF

(*Manual Pump*)
100:
	IF NOT Manual OR NOT Ready THEN
		OUT_LP   := 0;
		State    := 0;
	ELSE
		IF SI_Pump.Event = INIT_CONTINUOUS
		OR Event_Stop = INIT_CONTINUOUS
		THEN
			IF SoftStop THEN
				OUT_LP   := 0;
				State    := 0;
				RETURN;
			ELSE
				SoftStop := TRUE;
			END_IF
		END_IF

		IF SoftStop THEN
			EVP_Pump_Tgt := EVP_Pump_Tgt - CFG.EVP_Pump_Dec * CFG.Cycle;
			EVP_Pump_Tgt := MIN(EVP_Pump_Tgt, CFG.EVP_Pump_Max);
			EVP_Pump_Tgt := MIN(EVP_Pump_Tgt, IN_Hmi_Pump_Perc);
			EVP_Pump_Tgt := MAX(EVP_Pump_Tgt, CFG.EVP_Pump_Min);

			IF EVP_Pump_Tgt = CFG.EVP_Pump_Min OR CFG.EVP_Pump_Dec <= 0
			THEN EVP_Pump := 0;
			ELSE EVP_Pump := REAL_TO_UINT(EVP_Pump_Tgt * Perc * 10.0);
			END_IF

		ELSE
			EVP_Pump_Tgt := EVP_Pump_Tgt + CFG.EVP_Pump_Inc * CFG.Cycle;
			EVP_Pump_Tgt := MIN(EVP_Pump_Tgt, CFG.EVP_Pump_Max);
			EVP_Pump_Tgt := MIN(EVP_Pump_Tgt, IN_Hmi_Pump_Perc);
			EVP_Pump_Tgt := MAX(EVP_Pump_Tgt, CFG.EVP_Pump_Min);

			EVP_Pump := REAL_TO_UINT(EVP_Pump_Tgt * Perc * 10.0);

		END_IF

		IF EVP_Pump = 0 THEN
			OUT_LP   := 0;
			State    := 0; (*Next State*)
		ELSE
			OUT_LP   := 1;

		END_IF
	END_IF

(*****************************************************************************)
(** FILL                                                                    **)
(*****************************************************************************)
(*Port Fwd Fill - Open Valves*)
1010:
	IF Manual OR NOT Ready THEN
		State := 0;

	ELSIF TimeCnt > CFG.TimeMax_Init THEN
		Error := State;
		State := 0;

	ELSIF Event_Stop = INIT_CONTINUOUS OR Event_Dump = INIT_CONTINUOUS OR Event_Move = INIT_CONTINUOUS THEN
		WB_A.B_Open := FALSE;
		WB_E.B_Open := FALSE;
		WB_J.B_Open := FALSE;
		WB_L.B_Open := FALSE;

		TimeCnt := 0.0;
		State   := 5000;
		Next    := 0;

	ELSE
		IF Event_Fill = INIT_CONTINUOUS THEN
			Pause := NOT Pause;
		END_IF

		Init := TRUE;
	
		IF NOT (WB_A.SF_Open AND WB_A.State = 0) THEN WB_A.B_Open := TRUE; Init := FALSE; END_IF
		IF NOT (WB_E.SF_Open AND WB_E.State = 0) THEN WB_E.B_Open := TRUE; Init := FALSE; END_IF
		IF NOT (WB_J.SF_Open AND WB_J.State = 0) THEN WB_J.B_Open := TRUE; Init := FALSE; END_IF
		IF NOT (WB_L.SF_Open AND WB_L.State = 0) THEN WB_L.B_Open := TRUE; Init := FALSE; END_IF
	
		IF Init THEN
			WB_A.B_Open := FALSE;
			WB_E.B_Open := FALSE;
			WB_J.B_Open := FALSE;
			WB_L.B_Open := FALSE;

			State := 1100; (*Port Fill - Scoop Dw*)

		END_IF
	END_IF

(*Port Aft Fill - Open Valves*)
1020:
	IF Manual OR NOT Ready THEN
		State := 0;

	ELSIF TimeCnt > CFG.TimeMax_Init THEN
		Error := State;
		State := 0;

	ELSIF Event_Stop = INIT_CONTINUOUS OR Event_Dump = INIT_CONTINUOUS OR Event_Move = INIT_CONTINUOUS THEN
		WB_D.B_Open := FALSE;
		WB_E.B_Open := FALSE;
		WB_J.B_Open := FALSE;
		WB_L.B_Open := FALSE;

		TimeCnt := 0.0;
		State   := 5000;
		Next    := 0;

	ELSE
		IF Event_Fill = INIT_CONTINUOUS THEN
			Pause := NOT Pause;
		END_IF

		Init := TRUE;
	
		IF NOT (WB_D.SF_Open AND WB_D.State = 0) THEN WB_D.B_Open := TRUE; Init := FALSE; END_IF
		IF NOT (WB_E.SF_Open AND WB_E.State = 0) THEN WB_E.B_Open := TRUE; Init := FALSE; END_IF
		IF NOT (WB_J.SF_Open AND WB_J.State = 0) THEN WB_J.B_Open := TRUE; Init := FALSE; END_IF
		IF NOT (WB_L.SF_Open AND WB_L.State = 0) THEN WB_L.B_Open := TRUE; Init := FALSE; END_IF
	
		IF Init THEN
			WB_D.B_Open := FALSE;
			WB_E.B_Open := FALSE;
			WB_J.B_Open := FALSE;
			WB_L.B_Open := FALSE;

			State := 1100; (*Port Fill - Scoop Dw*)

		END_IF
	END_IF

(*Stbd Fwd Fill - Open Valves*)
1030:
	IF Manual OR NOT Ready THEN
		State := 0;

	ELSIF TimeCnt > CFG.TimeMax_Init THEN
		Error := State;
		State := 0;

	ELSIF Event_Stop = INIT_CONTINUOUS OR Event_Dump = INIT_CONTINUOUS OR Event_Move = INIT_CONTINUOUS THEN
		WB_F.B_Open := FALSE;
		WB_G.B_Open := FALSE;
		WB_H.B_Open := FALSE;
		WB_K.B_Open := FALSE;

		TimeCnt := 0.0;
		State   := 5000;
		Next    := 0;

	ELSE
		IF Event_Fill = INIT_CONTINUOUS THEN
			Pause := NOT Pause;
		END_IF

		Init := TRUE;
	
		IF NOT (WB_F.SF_Open AND WB_F.State = 0) THEN WB_F.B_Open := TRUE; Init := FALSE; END_IF
		IF NOT (WB_G.SF_Open AND WB_G.State = 0) THEN WB_G.B_Open := TRUE; Init := FALSE; END_IF
		IF NOT (WB_H.SF_Open AND WB_H.State = 0) THEN WB_H.B_Open := TRUE; Init := FALSE; END_IF
		IF NOT (WB_K.SF_Open AND WB_K.State = 0) THEN WB_K.B_Open := TRUE; Init := FALSE; END_IF
	
		IF Init THEN
			WB_F.B_Open := FALSE;
			WB_G.B_Open := FALSE;
			WB_H.B_Open := FALSE;
			WB_K.B_Open := FALSE;

			State := 1200; (*Stbd Fill - Scoop Dw*)

		END_IF
	END_IF

(*Stbd Aft Fill - Open Valves*)
1040:
	IF Manual OR NOT Ready THEN
		State := 0;

	ELSIF TimeCnt > CFG.TimeMax_Init THEN
		Error := State;
		State := 0;

	ELSIF Event_Stop = INIT_CONTINUOUS OR Event_Dump = INIT_CONTINUOUS OR Event_Move = INIT_CONTINUOUS THEN
		WB_F.B_Open := FALSE;
		WB_G.B_Open := FALSE;
		WB_H.B_Open := FALSE;
		WB_M.B_Open := FALSE;

		TimeCnt := 0.0;
		State   := 5000;
		Next    := 0;

	ELSE
		IF Event_Fill = INIT_CONTINUOUS THEN
			Pause := NOT Pause;
		END_IF

		Init := TRUE;
	
		IF NOT (WB_F.SF_Open AND WB_F.State = 0) THEN WB_F.B_Open := TRUE; Init := FALSE; END_IF
		IF NOT (WB_G.SF_Open AND WB_G.State = 0) THEN WB_G.B_Open := TRUE; Init := FALSE; END_IF
		IF NOT (WB_H.SF_Open AND WB_H.State = 0) THEN WB_H.B_Open := TRUE; Init := FALSE; END_IF
		IF NOT (WB_M.SF_Open AND WB_M.State = 0) THEN WB_M.B_Open := TRUE; Init := FALSE; END_IF

		IF Init THEN
			WB_F.B_Open := FALSE;
			WB_G.B_Open := FALSE;
			WB_H.B_Open := FALSE;
			WB_M.B_Open := FALSE;

			State := 1200; (*Stbd Fill - Scoop Dw*)

		END_IF
	END_IF

(*Port Fill - Stbd Scoop Dw*)
1100:
	IF Manual OR NOT Ready THEN
		State := 0;

	ELSIF TimeCnt > CFG.TimeMax_Init THEN
		Error := State;
		State := 0;

	ELSIF Event_Stop = INIT_CONTINUOUS OR Event_Dump = INIT_CONTINUOUS OR Event_Move = INIT_CONTINUOUS THEN
		WB_SUD.B_Half := FALSE;
		WB_SUD.B_Open := FALSE;

		TimeCnt := 0.0;
		State   := 5000;
		Next    := 0;

	ELSE
		IF Event_Fill = INIT_CONTINUOUS THEN
			Pause := NOT Pause;
		END_IF

		Init := TRUE;

		IF OUT_12
		THEN IF NOT (WB_SUD.SF_Half AND WB_SUD.State = 0) THEN WB_SUD.B_Half := TRUE; Init := FALSE; END_IF
		ELSE IF NOT (WB_SUD.SF_Open AND WB_SUD.State = 0) THEN WB_SUD.B_Open := TRUE; Init := FALSE; END_IF
		END_IF

		IF Init THEN
			WB_SUD.B_Half := FALSE;
			WB_SUD.B_Open := FALSE;

			EVP_Pump := REAL_TO_INT(EVP_Pump_Tgt * Perc * 10.0);
			OUT_LP   := 1;
			TimeCnt  := 0.0;
			State    := 1300;

		END_IF
	END_IF

(*Stbd Fill - Port Scoop Dw*)
1200:
	IF Manual OR NOT Ready THEN
		State := 0;

	ELSIF TimeCnt > CFG.TimeMax_Init THEN
		Error := State;
		State := 0;

	ELSIF Event_Stop = INIT_CONTINUOUS OR Event_Dump = INIT_CONTINUOUS OR Event_Move = INIT_CONTINUOUS THEN
		WB_PUD.B_Half := FALSE;
		WB_PUD.B_Open := FALSE;

		TimeCnt := 0.0;
		State   := 5000;
		Next    := 0;

	ELSE
		IF Event_Fill = INIT_CONTINUOUS THEN
			Pause := NOT Pause;
		END_IF

		Init := TRUE;

		IF OUT_12
		THEN IF NOT (WB_PUD.SF_Half AND WB_PUD.State = 0) THEN WB_PUD.B_Half := TRUE; Init := FALSE; END_IF
		ELSE IF NOT (WB_PUD.SF_Open AND WB_PUD.State = 0) THEN WB_PUD.B_Open := TRUE; Init := FALSE; END_IF
		END_IF

		IF Init THEN
			WB_PUD.B_Half := FALSE;
			WB_PUD.B_Open := FALSE;

			EVP_Pump := REAL_TO_INT(EVP_Pump_Tgt * Perc * 10.0);
			OUT_LP   := 1;
			TimeCnt  := 0.0;
			State    := 1300;

		END_IF
	END_IF

(*Fill Pump*)
1300:
	IF Manual OR NOT Ready THEN
		OUT_LP   := 0;
		State    := 0;

	ELSE
		IF Event_Stop = INIT_CONTINUOUS OR Event_Dump = INIT_CONTINUOUS OR Event_Move = INIT_CONTINUOUS THEN
			SoftStop := TRUE;
		END_IF

		IF Event_Fill = INIT_CONTINUOUS THEN
			Pause := NOT Pause;
		END_IF

		IF SoftStop OR Pause THEN
			EVP_Pump_Tgt := EVP_Pump_Tgt - CFG.EVP_Pump_Dec * CFG.Cycle;
			EVP_Pump_Tgt := MIN(EVP_Pump_Tgt, CFG.EVP_Pump_Max);
			EVP_Pump_Tgt := MAX(EVP_Pump_Tgt, CFG.EVP_Pump_Min);

			IF EVP_Pump_Tgt = CFG.EVP_Pump_Min OR CFG.EVP_Pump_Dec <= 0
			THEN EVP_Pump := 0;
			ELSE EVP_Pump := REAL_TO_UINT(EVP_Pump_Tgt * Perc * 10.0);
			END_IF

		ELSE
			EVP_Pump_Tgt := EVP_Pump_Tgt + CFG.EVP_Pump_Inc * CFG.Cycle;
			EVP_Pump_Tgt := MIN(EVP_Pump_Tgt, CFG.EVP_Pump_Max);
			EVP_Pump_Tgt := MAX(EVP_Pump_Tgt, CFG.EVP_Pump_Min);

			EVP_Pump := REAL_TO_UINT(EVP_Pump_Tgt * Perc * 10.0);

		END_IF

		IF EVP_Pump = 0 THEN
			OUT_LP := 0;

			IF SoftStop THEN
				TimeCnt := 0.0;
				State   := 5000;
				Next    := 0;
			END_IF

		ELSE
			OUT_LP := 1;

		END_IF
	END_IF

(*****************************************************************************)
(** DUMP                                                                    **)
(*****************************************************************************)
(*Port DUMP - Stbd Scoop Aft / Dw*)
2010,2020:
	IF Manual OR NOT Ready THEN
		State := 0;

	ELSIF TimeCnt > CFG.TimeMax_Init THEN
		Error := State;
		State := 0;

	ELSIF Event_Stop = INIT_CONTINUOUS OR Event_Fill = INIT_CONTINUOUS OR Event_Move = INIT_CONTINUOUS THEN
		WB_SAF.B_Open := FALSE;
		WB_SUD.B_Half := FALSE;
		WB_SUD.B_Open := FALSE;

		TimeCnt := 0.0;
		State   := 5000;
		Next    := 0;

	ELSE
		IF Event_Dump = INIT_CONTINUOUS THEN
			Pause := NOT Pause;
		END_IF

		Init := TRUE;

		IF CFG.EnScoopAF
		THEN IF NOT (WB_SAF.SF_Open AND WB_SAF.State = 0) THEN WB_SAF.B_Open := TRUE; Init := FALSE; END_IF
		END_IF

		IF OUT_12
		THEN IF NOT (WB_SUD.SF_Half AND WB_SUD.State = 0) THEN WB_SUD.B_Half := TRUE; Init := FALSE; END_IF
		ELSE IF NOT (WB_SUD.SF_Open AND WB_SUD.State = 0) THEN WB_SUD.B_Open := TRUE; Init := FALSE; END_IF
		END_IF

		IF Init THEN
			WB_SAF.B_Open := FALSE;
			WB_SUD.B_Half := FALSE;
			WB_SUD.B_Open := FALSE;

			State := State + 200; (*Dump Pump Valves*)

		END_IF
	END_IF

(*Stbd DUMP - Port Scoop Aft / Dw*)
2030,2040:
	IF Manual OR NOT Ready THEN
		State := 0;

	ELSIF TimeCnt > CFG.TimeMax_Init THEN
		Error := State;
		State := 0;

	ELSIF Event_Stop = INIT_CONTINUOUS OR Event_Fill = INIT_CONTINUOUS OR Event_Move = INIT_CONTINUOUS THEN
		WB_PAF.B_Open := FALSE;
		WB_PUD.B_Half := FALSE;
		WB_PUD.B_Open := FALSE;

		TimeCnt := 0.0;
		State   := 5000;
		Next    := 0;

	ELSE
		IF Event_Dump = INIT_CONTINUOUS THEN
			Pause := NOT Pause;
		END_IF

		Init := TRUE;
	
		IF CFG.EnScoopAF
		THEN IF NOT (WB_PAF.SF_Open AND WB_PAF.State = 0) THEN WB_PAF.B_Open := TRUE; Init := FALSE; END_IF
		END_IF

		IF OUT_12 (*Test3*)
		THEN IF NOT (WB_PUD.SF_Half AND WB_PUD.State = 0) THEN WB_PUD.B_Half := TRUE; Init := FALSE; END_IF
		ELSE IF NOT (WB_PUD.SF_Open AND WB_PUD.State = 0) THEN WB_PUD.B_Open := TRUE; Init := FALSE; END_IF
		END_IF

		IF Init THEN
			WB_PAF.B_Open := FALSE;
			WB_PUD.B_Half := FALSE;
			WB_PUD.B_Open := FALSE;

			State := State + 200; (*Dump Pump Valves*)

		END_IF
	END_IF

(*Port Fwd Dump - Valves*)
2210:
	IF Manual OR NOT Ready THEN
		State := 0;

	ELSIF TimeCnt > CFG.TimeMax_Init THEN
		Error := State;
		State := 0;

	ELSIF Event_Stop = INIT_CONTINUOUS OR Event_Fill = INIT_CONTINUOUS OR Event_Move = INIT_CONTINUOUS THEN
		WB_A.B_Open := FALSE;
		WB_F.B_Open := FALSE;
		WB_H.B_Open := FALSE;
		WB_J.B_Open := FALSE;

		TimeCnt := 0.0;
		State   := 5000;
		Next    := 0;

	ELSE
		IF Event_Dump = INIT_CONTINUOUS THEN
			Pause := NOT Pause;
		END_IF

		Init := TRUE;
	
		IF NOT (WB_A.SF_Open AND WB_A.State = 0) THEN WB_A.B_Open := TRUE; Init := FALSE; END_IF
		IF NOT (WB_F.SF_Open AND WB_F.State = 0) THEN WB_F.B_Open := TRUE; Init := FALSE; END_IF
		IF NOT (WB_H.SF_Open AND WB_H.State = 0) THEN WB_H.B_Open := TRUE; Init := FALSE; END_IF
		IF NOT (WB_J.SF_Open AND WB_J.State = 0) THEN WB_J.B_Open := TRUE; Init := FALSE; END_IF
	
		IF Init THEN
			WB_A.B_Open := FALSE;
			WB_F.B_Open := FALSE;
			WB_H.B_Open := FALSE;
			WB_J.B_Open := FALSE;

			TimeCnt  := 0.0;

			IF SF_P_Fwd THEN
				State := State + 200; (*if already empty jump pump*)
			ELSE
				EVP_Pump := REAL_TO_INT(EVP_Pump_Tgt * Perc * 10.0);
				OUT_LP   := 1;
				State    := State + 100; (*Port Fwd Dump - Pump*)
			END_IF

		END_IF
	END_IF

(*Port Aft Dump - Valves*)
2220:
	IF Manual OR NOT Ready THEN
		State := 0;

	ELSIF TimeCnt > CFG.TimeMax_Init THEN
		Error := State;
		State := 0;

	ELSIF Event_Stop = INIT_CONTINUOUS OR Event_Fill = INIT_CONTINUOUS OR Event_Move = INIT_CONTINUOUS THEN
		WB_D.B_Open := FALSE;
		WB_F.B_Open := FALSE;
		WB_H.B_Open := FALSE;
		WB_J.B_Open := FALSE;

		TimeCnt := 0.0;
		State   := 5000;
		Next    := 0;

	ELSE
		IF Event_Dump = INIT_CONTINUOUS THEN
			Pause := NOT Pause;
		END_IF

		Init := TRUE;
	
		IF NOT (WB_D.SF_Open AND WB_D.State = 0) THEN WB_D.B_Open := TRUE; Init := FALSE; END_IF
		IF NOT (WB_F.SF_Open AND WB_F.State = 0) THEN WB_F.B_Open := TRUE; Init := FALSE; END_IF
		IF NOT (WB_H.SF_Open AND WB_H.State = 0) THEN WB_H.B_Open := TRUE; Init := FALSE; END_IF
		IF NOT (WB_J.SF_Open AND WB_J.State = 0) THEN WB_J.B_Open := TRUE; Init := FALSE; END_IF
	
		IF Init THEN
			WB_D.B_Open := FALSE;
			WB_F.B_Open := FALSE;
			WB_H.B_Open := FALSE;
			WB_J.B_Open := FALSE;

			TimeCnt  := 0.0;

			IF SF_P_Aft THEN
				State := State + 200; (*if already empty jumo pump*)
			ELSE
				EVP_Pump := REAL_TO_INT(EVP_Pump_Tgt * Perc * 10.0);
				OUT_LP   := 1;
				State    := State + 100; (*Port Fwd Dump - Pump*)
			END_IF

		END_IF
	END_IF

(*Stbd Fwd Dump - Valves*)
2230:
	IF Manual OR NOT Ready THEN
		State := 0;

	ELSIF TimeCnt > CFG.TimeMax_Init THEN
		Error := State;
		State := 0;

	ELSIF Event_Stop = INIT_CONTINUOUS OR Event_Fill = INIT_CONTINUOUS OR Event_Move = INIT_CONTINUOUS THEN
		WB_E.B_Open := FALSE;
		WB_G.B_Open := FALSE;
		WB_K.B_Open := FALSE;
		WB_L.B_Open := FALSE;

		TimeCnt := 0.0;
		State   := 5000;
		Next    := 0;

	ELSE
		IF Event_Dump = INIT_CONTINUOUS THEN
			Pause := NOT Pause;
		END_IF

		Init := TRUE;

		IF NOT (WB_E.SF_Open AND WB_E.State = 0) THEN WB_E.B_Open := TRUE; Init := FALSE; END_IF
		IF NOT (WB_G.SF_Open AND WB_G.State = 0) THEN WB_G.B_Open := TRUE; Init := FALSE; END_IF
		IF NOT (WB_K.SF_Open AND WB_K.State = 0) THEN WB_K.B_Open := TRUE; Init := FALSE; END_IF
		IF NOT (WB_L.SF_Open AND WB_L.State = 0) THEN WB_L.B_Open := TRUE; Init := FALSE; END_IF
	
		IF Init THEN
			WB_E.B_Open := FALSE;
			WB_G.B_Open := FALSE;
			WB_K.B_Open := FALSE;
			WB_L.B_Open := FALSE;

			TimeCnt  := 0.0;

			IF SF_S_Fwd THEN
				State := State + 200; (*if already empty jumo pump*)
			ELSE
				EVP_Pump := REAL_TO_INT(EVP_Pump_Tgt * Perc * 10.0);
				OUT_LP   := 1;
				State    := State + 100; (*Port Fwd Dump - Pump*)
			END_IF

		END_IF
	END_IF


(*Stbd Aft Dump - Valves*)
2240:
	IF Manual OR NOT Ready THEN
		State := 0;

	ELSIF TimeCnt > CFG.TimeMax_Init THEN
		Error := State;
		State := 0;

	ELSIF Event_Stop = INIT_CONTINUOUS OR Event_Fill = INIT_CONTINUOUS OR Event_Move = INIT_CONTINUOUS THEN
		WB_E.B_Open := FALSE;
		WB_G.B_Open := FALSE;
		WB_M.B_Open := FALSE;
		WB_L.B_Open := FALSE;

		TimeCnt := 0.0;
		State   := 5000;
		Next    := 0;

	ELSE
		IF Event_Dump = INIT_CONTINUOUS THEN
			Pause := NOT Pause;
		END_IF

		Init := TRUE;
	
		IF NOT (WB_E.SF_Open AND WB_E.State = 0) THEN WB_E.B_Open := TRUE; Init := FALSE; END_IF
		IF NOT (WB_G.SF_Open AND WB_G.State = 0) THEN WB_G.B_Open := TRUE; Init := FALSE; END_IF
		IF NOT (WB_M.SF_Open AND WB_M.State = 0) THEN WB_M.B_Open := TRUE; Init := FALSE; END_IF
		IF NOT (WB_L.SF_Open AND WB_L.State = 0) THEN WB_L.B_Open := TRUE; Init := FALSE; END_IF
	
		IF Init THEN
			WB_E.B_Open := FALSE;
			WB_G.B_Open := FALSE;
			WB_M.B_Open := FALSE;
			WB_L.B_Open := FALSE;

			TimeCnt  := 0.0;

			IF SF_S_Aft THEN
				State := State + 200; (*if already empty jump pump*)
			ELSE
				EVP_Pump := REAL_TO_INT(EVP_Pump_Tgt * Perc * 10.0);
				OUT_LP   := 1;
				State    := State + 100; (*Port Fwd Dump - Pump*)
			END_IF

		END_IF
	END_IF

(*DUMP Pump*)
2310,2320,2330,2340:
	IF Manual OR NOT Ready THEN
		OUT_LP   := 0;
		State    := 0;

	ELSE
		IF Event_Stop = INIT_CONTINUOUS OR Event_Fill = INIT_CONTINUOUS OR Event_Move = INIT_CONTINUOUS
		OR State = 2310 AND SF_P_Fwd
		OR State = 2320 AND SF_P_Aft
		OR State = 2330 AND SF_S_Fwd
		OR State = 2340 AND SF_S_Aft
		THEN
			SoftStop := TRUE;
		END_IF

		IF Event_Dump = INIT_CONTINUOUS THEN
			Pause := NOT Pause;
		END_IF

		IF SoftStop OR Pause THEN
			EVP_Pump_Tgt := EVP_Pump_Tgt - CFG.EVP_Pump_Dec * CFG.Cycle;
			EVP_Pump_Tgt := MIN(EVP_Pump_Tgt, CFG.EVP_Pump_Max);
			EVP_Pump_Tgt := MAX(EVP_Pump_Tgt, CFG.EVP_Pump_Min);

			IF EVP_Pump_Tgt = CFG.EVP_Pump_Min OR CFG.EVP_Pump_Dec <= 0
			THEN EVP_Pump := 0;
			ELSE EVP_Pump := REAL_TO_UINT(EVP_Pump_Tgt * Perc * 10.0);
			END_IF

		ELSE
			EVP_Pump_Tgt := EVP_Pump_Tgt + CFG.EVP_Pump_Inc * CFG.Cycle;
			EVP_Pump_Tgt := MIN(EVP_Pump_Tgt, CFG.EVP_Pump_Max);
			EVP_Pump_Tgt := MAX(EVP_Pump_Tgt, CFG.EVP_Pump_Min);

			EVP_Pump := REAL_TO_UINT(EVP_Pump_Tgt * Perc * 10.0);

		END_IF

		IF EVP_Pump = 0 THEN
			OUT_LP := 0;

			IF SoftStop THEN
				TimeCnt := 0.0;
				State   := State + 100;
			END_IF

		ELSE
			OUT_LP := 1;

		END_IF
	END_IF

(*Port Dump - Valves2*)
2410,2420:
	IF Manual OR NOT Ready THEN
		State := 0;

	ELSIF TimeCnt > CFG.TimeMax_Init THEN
		Error := State;
		State := 0;

	ELSIF Event_Stop = INIT_CONTINUOUS OR Event_Fill = INIT_CONTINUOUS OR Event_Move = INIT_CONTINUOUS THEN
		WB_E.B_Open  := FALSE;
		WB_F.B_Close := FALSE;

		TimeCnt := 0.0;
		State   := 5000;
		Next    := 0;

	ELSE
		Init := TRUE;
	
		IF NOT (WB_E.SF_Open  AND WB_E.State = 0) THEN WB_E.B_Open  := TRUE; Init := FALSE; END_IF
		IF NOT (WB_F.SF_Close AND WB_F.State = 0) THEN WB_F.B_Close := TRUE; Init := FALSE; END_IF

		IF Init THEN
			WB_E.B_Open  := FALSE;
			WB_F.B_Close := FALSE;

			TimeCnt  := 0.0;
			State    := 2500; (*Port Dump*)

		END_IF
	END_IF

(*Stbd Dump - Valves2*)
2430,2440:
	IF Manual OR NOT Ready THEN
		State := 0;

	ELSIF TimeCnt > CFG.TimeMax_Init THEN
		Error := State;
		State := 0;

	ELSIF Event_Stop = INIT_CONTINUOUS OR Event_Fill = INIT_CONTINUOUS OR Event_Move = INIT_CONTINUOUS THEN
		WB_H.B_Open  := FALSE;
		WB_L.B_Close := FALSE;

		TimeCnt := 0.0;
		State   := 5000;
		Next    := 0;

	ELSE
		Init := TRUE;
	
		IF NOT (WB_H.SF_Open  AND WB_H.State = 0) THEN WB_H.B_Open  := TRUE; Init := FALSE; END_IF
		IF NOT (WB_L.SF_Close AND WB_L.State = 0) THEN WB_L.B_Close := TRUE; Init := FALSE; END_IF

		IF Init THEN
			WB_H.B_Open  := FALSE;
			WB_L.B_Close := FALSE;

			TimeCnt  := 0.0;
			State    := 2500; (*Port Dump*)

		END_IF
	END_IF

(*DUMP - WAIT*)
2500:
	IF Manual OR NOT Ready THEN
		State := 0;

	ELSIF TimeCnt > TimeDump OR Event_Stop = INIT_CONTINUOUS OR Event_Fill = INIT_CONTINUOUS OR Event_Move = INIT_CONTINUOUS THEN
		TimeCnt := 0.0;
		State   := 5000;
		Next    := 0;

	END_IF

(*****************************************************************************)
(** MOVE                                                                    **)
(*****************************************************************************)
(*Port Fwd Move - Open Valves*)
3010:
	IF Manual OR NOT Ready THEN
		State := 0;

	ELSIF TimeCnt > CFG.TimeMax_Init THEN
		Error := State;
		State := 0;

	ELSIF Event_Stop = INIT_CONTINUOUS OR Event_Dump = INIT_CONTINUOUS OR Event_Fill = INIT_CONTINUOUS THEN
		WB_C.B_Open := FALSE;
		WB_S.B_Open := FALSE;

		TimeCnt := 0.0;
		State   := 5000;
		Next    := 0;

	ELSE
		IF Event_Move = INIT_CONTINUOUS THEN
			Pause := NOT Pause;
		END_IF

		Init := TRUE;
	
		IF NOT (WB_C.SF_Open AND WB_C.State = 0) THEN WB_C.B_Open := TRUE; Init := FALSE; END_IF
		IF NOT (WB_S.SF_Open AND WB_S.State = 0) THEN WB_S.B_Open := TRUE; Init := FALSE; END_IF

		IF Init THEN
			WB_C.B_Open := FALSE;
			WB_S.B_Open := FALSE;

			State := State + 100;

		END_IF
	END_IF

(*Port Aft Move - Open Valves*)
3020:
	IF Manual OR NOT Ready THEN
		State := 0;

	ELSIF TimeCnt > CFG.TimeMax_Init THEN
		Error := State;
		State := 0;

	ELSIF Event_Stop = INIT_CONTINUOUS OR Event_Dump = INIT_CONTINUOUS OR Event_Fill = INIT_CONTINUOUS THEN
		WB_B.B_Open := FALSE;

		TimeCnt := 0.0;
		State   := 5000;
		Next    := 0;

	ELSE
		IF Event_Move = INIT_CONTINUOUS THEN
			Pause := NOT Pause;
		END_IF

		Init := TRUE;
	
		IF NOT (WB_B.SF_Open AND WB_B.State = 0) THEN WB_B.B_Open := TRUE; Init := FALSE; END_IF

		IF Init THEN
			WB_B.B_Open := FALSE;

			State := State + 100;

		END_IF
	END_IF

(*Stbd Fwd Move - Open Valves*)
3030:
	IF Manual OR NOT Ready THEN
		State := 0;

	ELSIF TimeCnt > CFG.TimeMax_Init THEN
		Error := State;
		State := 0;

	ELSIF Event_Stop = INIT_CONTINUOUS OR Event_Dump = INIT_CONTINUOUS OR Event_Fill = INIT_CONTINUOUS THEN
		WB_N.B_Open := FALSE;
		WB_R.B_Open := FALSE;

		TimeCnt := 0.0;
		State   := 5000;
		Next    := 0;

	ELSE
		IF Event_Move = INIT_CONTINUOUS THEN
			Pause := NOT Pause;
		END_IF

		Init := TRUE;
	
		IF NOT (WB_N.SF_Open AND WB_N.State = 0) THEN WB_N.B_Open := TRUE; Init := FALSE; END_IF
		IF NOT (WB_R.SF_Open AND WB_R.State = 0) THEN WB_R.B_Open := TRUE; Init := FALSE; END_IF

		IF Init THEN
			WB_N.B_Open := FALSE;
			WB_R.B_Open := FALSE;

			State := State + 100;

		END_IF
	END_IF

(*Stbd Aft Move - Open Valves*)
3040:
	IF Manual OR NOT Ready THEN
		State := 0;

	ELSIF TimeCnt > CFG.TimeMax_Init THEN
		Error := State;
		State := 0;

	ELSIF Event_Stop = INIT_CONTINUOUS OR Event_Dump = INIT_CONTINUOUS OR Event_Fill = INIT_CONTINUOUS THEN
		WB_I.B_Open := FALSE;

		TimeCnt := 0.0;
		State   := 5000;
		Next    := 0;

	ELSE
		IF Event_Move = INIT_CONTINUOUS THEN
			Pause := NOT Pause;
		END_IF

		Init := TRUE;
	
		IF NOT (WB_I.SF_Open AND WB_I.State = 0) THEN WB_I.B_Open := TRUE; Init := FALSE; END_IF

		IF Init THEN
			WB_I.B_Open := FALSE;

			State := State + 100;

		END_IF
	END_IF

(*Port Fwd Move - Open Valves2*)
3110:
	IF Manual OR NOT Ready THEN
		State := 0;

	ELSIF TimeCnt > CFG.TimeMax_Init THEN
		Error := State;
		State := 0;

	ELSIF Event_Stop = INIT_CONTINUOUS OR Event_Dump = INIT_CONTINUOUS OR Event_Fill = INIT_CONTINUOUS THEN
		WB_N.B_Open := FALSE;
		WB_R.B_Open := FALSE;

		TimeCnt := 0.0;
		State   := 5000;
		Next    := 0;

	ELSE
		IF Event_Move = INIT_CONTINUOUS THEN
			Pause := NOT Pause;
		END_IF

		Init := TRUE;
	
		IF NOT (WB_N.SF_Open AND WB_N.State = 0) THEN WB_N.B_Open := TRUE; Init := FALSE; END_IF
		IF NOT (WB_R.SF_Open AND WB_R.State = 0) THEN WB_R.B_Open := TRUE; Init := FALSE; END_IF

		IF Init THEN
			WB_N.B_Open := FALSE;
			WB_R.B_Open := FALSE;

			TimeCnt  := 0.0;
			State := State + 100;

		END_IF
	END_IF

(*Port Aft Move - Open Valves2*)
3120:
	IF Manual OR NOT Ready THEN
		State := 0;

	ELSIF TimeCnt > CFG.TimeMax_Init THEN
		Error := State;
		State := 0;

	ELSIF Event_Stop = INIT_CONTINUOUS OR Event_Dump = INIT_CONTINUOUS OR Event_Fill = INIT_CONTINUOUS THEN
		WB_I.B_Open := FALSE;

		TimeCnt := 0.0;
		State   := 5000;
		Next    := 0;

	ELSE
		IF Event_Move = INIT_CONTINUOUS THEN
			Pause := NOT Pause;
		END_IF

		Init := TRUE;
	
		IF NOT (WB_I.SF_Open AND WB_I.State = 0) THEN WB_I.B_Open := TRUE; Init := FALSE; END_IF

		IF Init THEN
			WB_I.B_Open := FALSE;

			TimeCnt  := 0.0;
			State := State + 100;

		END_IF
	END_IF

(*Stbd Fwd Move - Open Valves2*)
3130:
	IF Manual OR NOT Ready THEN
		State := 0;

	ELSIF TimeCnt > CFG.TimeMax_Init THEN
		Error := State;
		State := 0;

	ELSIF Event_Stop = INIT_CONTINUOUS OR Event_Dump = INIT_CONTINUOUS OR Event_Fill = INIT_CONTINUOUS THEN
		WB_C.B_Open := FALSE;
		WB_S.B_Open := FALSE;

		TimeCnt := 0.0;
		State   := 5000;
		Next    := 0;

	ELSE
		IF Event_Move = INIT_CONTINUOUS THEN
			Pause := NOT Pause;
		END_IF

		Init := TRUE;
	
		IF NOT (WB_C.SF_Open AND WB_C.State = 0) THEN WB_C.B_Open := TRUE; Init := FALSE; END_IF
		IF NOT (WB_S.SF_Open AND WB_S.State = 0) THEN WB_S.B_Open := TRUE; Init := FALSE; END_IF

		IF Init THEN
			WB_C.B_Open := FALSE;
			WB_S.B_Open := FALSE;

			TimeCnt  := 0.0;
			State := State + 100;

		END_IF
	END_IF

(*Stbd Aft Move - Open Valves2*)
3140:
	IF Manual OR NOT Ready THEN
		State := 0;

	ELSIF TimeCnt > CFG.TimeMax_Init THEN
		Error := State;
		State := 0;

	ELSIF Event_Stop = INIT_CONTINUOUS OR Event_Dump = INIT_CONTINUOUS OR Event_Fill = INIT_CONTINUOUS THEN
		WB_B.B_Open := FALSE;

		TimeCnt := 0.0;
		State   := 5000;
		Next    := 0;

	ELSE
		IF Event_Move = INIT_CONTINUOUS THEN
			Pause := NOT Pause;
		END_IF

		Init := TRUE;
	
		IF NOT (WB_B.SF_Open AND WB_B.State = 0) THEN WB_B.B_Open := TRUE; Init := FALSE; END_IF

		IF Init THEN
			WB_B.B_Open := FALSE;

			TimeCnt  := 0.0;
			State := State + 100;

		END_IF
	END_IF

(*Move - WAIT BEFORE PUMP*)
3210,3220,3230,3240:
	IF Manual OR NOT Ready THEN
		State := 0;

	ELSIF Event_Dump = INIT_CONTINUOUS OR Event_Fill = INIT_CONTINUOUS THEN
		TimeCnt := 0.0;
		State   := 5000;
		Next    := 0;

	ELSE
		IF Event_Move = INIT_CONTINUOUS THEN
			Pause := NOT Pause;
		END_IF

		IF Event_Stop = INIT_CONTINUOUS OR TimeCnt > TimeMove THEN
			TimeCnt := 0.0;
			State   := State + 100;
		END_IF

	END_IF

(*Port Fwd Move - Close Valves2*)
3310:
	IF Manual OR NOT Ready THEN
		State := 0;

	ELSIF TimeCnt > CFG.TimeMax_Init THEN
		Error := State;
		State := 0;

	ELSIF Event_Stop = INIT_CONTINUOUS OR Event_Dump = INIT_CONTINUOUS OR Event_Fill = INIT_CONTINUOUS THEN
		WB_N.B_Close := FALSE;
		WB_R.B_Close := FALSE;

		TimeCnt := 0.0;
		State   := 5000;
		Next    := 0;

	ELSE
		IF Event_Move = INIT_CONTINUOUS THEN
			Pause := NOT Pause;
		END_IF

		Init := TRUE;

		IF NOT (WB_N.SF_Close AND WB_N.State = 0) THEN WB_N.B_Close := TRUE; Init := FALSE; END_IF
		IF NOT (WB_R.SF_Close AND WB_R.State = 0) THEN WB_R.B_Close := TRUE; Init := FALSE; END_IF

		IF Init THEN
			WB_N.B_Close := FALSE;
			WB_R.B_Close := FALSE;

			State := State + 100;

		END_IF
	END_IF

(*Port Aft Move - Close Valves2*)
3320:
	IF Manual OR NOT Ready THEN
		State := 0;

	ELSIF TimeCnt > CFG.TimeMax_Init THEN
		Error := State;
		State := 0;

	ELSIF Event_Stop = INIT_CONTINUOUS OR Event_Dump = INIT_CONTINUOUS OR Event_Fill = INIT_CONTINUOUS THEN
		WB_I.B_Close := FALSE;

		TimeCnt := 0.0;
		State   := 5000;
		Next    := 0;

	ELSE
		IF Event_Move = INIT_CONTINUOUS THEN
			Pause := NOT Pause;
		END_IF

		Init := TRUE;
	
		IF NOT (WB_I.SF_Close AND WB_I.State = 0) THEN WB_I.B_Close := TRUE; Init := FALSE; END_IF

		IF Init THEN
			WB_I.B_Close := FALSE;

			State := State + 100;

		END_IF
	END_IF

(*Stbd Fwd Move - Close Valves2*)
3330:
	IF Manual OR NOT Ready THEN
		State := 0;

	ELSIF TimeCnt > CFG.TimeMax_Init THEN
		Error := State;
		State := 0;

	ELSIF Event_Stop = INIT_CONTINUOUS OR Event_Dump = INIT_CONTINUOUS OR Event_Fill = INIT_CONTINUOUS THEN
		WB_C.B_Close := FALSE;
		WB_S.B_Close := FALSE;

		TimeCnt := 0.0;
		State   := 5000;
		Next    := 0;

	ELSE
		IF Event_Move = INIT_CONTINUOUS THEN
			Pause := NOT Pause;
		END_IF

		Init := TRUE;
	
		IF NOT (WB_C.SF_Close AND WB_C.State = 0) THEN WB_C.B_Close := TRUE; Init := FALSE; END_IF
		IF NOT (WB_S.SF_Close AND WB_S.State = 0) THEN WB_S.B_Close := TRUE; Init := FALSE; END_IF

		IF Init THEN
			WB_C.B_Close := FALSE;
			WB_S.B_Close := FALSE;

			State := State + 100;

		END_IF
	END_IF

(*Stbd Aft Move - Close Valves2*)
3340:
	IF Manual OR NOT Ready THEN
		State := 0;

	ELSIF TimeCnt > CFG.TimeMax_Init THEN
		Error := State;
		State := 0;

	ELSIF Event_Stop = INIT_CONTINUOUS OR Event_Dump = INIT_CONTINUOUS OR Event_Fill = INIT_CONTINUOUS THEN
		WB_B.B_Close := FALSE;

		TimeCnt := 0.0;
		State   := 5000;
		Next    := 0;

	ELSE
		IF Event_Move = INIT_CONTINUOUS THEN
			Pause := NOT Pause;
		END_IF

		Init := TRUE;
	
		IF NOT (WB_B.SF_Close AND WB_B.State = 0) THEN WB_B.B_Close := TRUE; Init := FALSE; END_IF

		IF Init THEN
			WB_B.B_Close := FALSE;

			State := State + 100;

		END_IF
	END_IF

(*Port Fwd Move - Close Valves*)
3410:
	IF Manual OR NOT Ready THEN
		State := 0;

	ELSIF TimeCnt > CFG.TimeMax_Init THEN
		Error := State;
		State := 0;

	ELSIF Event_Stop = INIT_CONTINUOUS OR Event_Dump = INIT_CONTINUOUS OR Event_Fill = INIT_CONTINUOUS THEN
		WB_C.B_Close := FALSE;
		WB_S.B_Close := FALSE;

		TimeCnt := 0.0;
		State   := 5000;
		Next    := 0;

	ELSE
		IF Event_Move = INIT_CONTINUOUS THEN
			Pause := NOT Pause;
		END_IF

		Init := TRUE;
	
		IF NOT (WB_C.SF_Close AND WB_C.State = 0) THEN WB_C.B_Close := TRUE; Init := FALSE; END_IF
		IF NOT (WB_S.SF_Close AND WB_S.State = 0) THEN WB_S.B_Close := TRUE; Init := FALSE; END_IF

		IF Init THEN
			WB_C.B_Close := FALSE;
			WB_S.B_Close := FALSE;

			State := State + 100;

		END_IF
	END_IF

(*Port Aft Move - Close Valves*)
3420:
	IF Manual OR NOT Ready THEN
		State := 0;

	ELSIF TimeCnt > CFG.TimeMax_Init THEN
		Error := State;
		State := 0;

	ELSIF Event_Stop = INIT_CONTINUOUS OR Event_Dump = INIT_CONTINUOUS OR Event_Fill = INIT_CONTINUOUS THEN
		WB_B.B_Close := FALSE;

		TimeCnt := 0.0;
		State   := 5000;
		Next    := 0;

	ELSE
		IF Event_Move = INIT_CONTINUOUS THEN
			Pause := NOT Pause;
		END_IF

		Init := TRUE;
	
		IF NOT (WB_B.SF_Close AND WB_B.State = 0) THEN WB_B.B_Close := TRUE; Init := FALSE; END_IF

		IF Init THEN
			WB_B.B_Close := FALSE;

			State := State + 100;

		END_IF
	END_IF

(*Stbd Fwd Move - Close Valves*)
3430:
	IF Manual OR NOT Ready THEN
		State := 0;

	ELSIF TimeCnt > CFG.TimeMax_Init THEN
		Error := State;
		State := 0;

	ELSIF Event_Stop = INIT_CONTINUOUS OR Event_Dump = INIT_CONTINUOUS OR Event_Fill = INIT_CONTINUOUS THEN
		WB_N.B_Close := FALSE;
		WB_R.B_Close := FALSE;

		TimeCnt := 0.0;
		State   := 5000;
		Next    := 0;

	ELSE
		IF Event_Move = INIT_CONTINUOUS THEN
			Pause := NOT Pause;
		END_IF

		Init := TRUE;
	
		IF NOT (WB_N.SF_Close AND WB_N.State = 0) THEN WB_N.B_Close := TRUE; Init := FALSE; END_IF
		IF NOT (WB_R.SF_Close AND WB_R.State = 0) THEN WB_R.B_Close := TRUE; Init := FALSE; END_IF

		IF Init THEN
			WB_N.B_Close := FALSE;
			WB_R.B_Close := FALSE;

			State := State + 100;

		END_IF
	END_IF

(*Stbd Aft Move - Close Valves*)
3440:
	IF Manual OR NOT Ready THEN
		State := 0;

	ELSIF TimeCnt > CFG.TimeMax_Init THEN
		Error := State;
		State := 0;

	ELSIF Event_Stop = INIT_CONTINUOUS OR Event_Dump = INIT_CONTINUOUS OR Event_Fill = INIT_CONTINUOUS THEN
		WB_I.B_Close := FALSE;

		TimeCnt := 0.0;
		State   := 5000;
		Next    := 0;

	ELSE
		IF Event_Move = INIT_CONTINUOUS THEN
			Pause := NOT Pause;
		END_IF

		Init := TRUE;
	
		IF NOT (WB_I.SF_Close AND WB_I.State = 0) THEN WB_I.B_Close := TRUE; Init := FALSE; END_IF

		IF Init THEN
			WB_I.B_Close := FALSE;

			State := State + 100;

		END_IF
	END_IF

(*Port Fwd Move - Open Valves3*)
3510:
	IF Manual OR NOT Ready THEN
		State := 0;

	ELSIF TimeCnt > CFG.TimeMax_Init THEN
		Error := State;
		State := 0;

	ELSIF Event_Stop = INIT_CONTINUOUS OR Event_Dump = INIT_CONTINUOUS OR Event_Fill = INIT_CONTINUOUS THEN
		WB_A.B_Open := FALSE;
		WB_E.B_Open := FALSE;
		WB_K.B_Open := FALSE;
		WB_L.B_Open := FALSE;

		TimeCnt := 0.0;
		State   := 5000;
		Next    := 0;

	ELSE
		IF Event_Move = INIT_CONTINUOUS THEN
			Pause := NOT Pause;
		END_IF

		Init := TRUE;
	
		IF NOT (WB_A.SF_Open AND WB_A.State = 0) THEN WB_A.B_Open := TRUE; Init := FALSE; END_IF
		IF NOT (WB_E.SF_Open AND WB_E.State = 0) THEN WB_E.B_Open := TRUE; Init := FALSE; END_IF
		IF NOT (WB_K.SF_Open AND WB_K.State = 0) THEN WB_K.B_Open := TRUE; Init := FALSE; END_IF
		IF NOT (WB_L.SF_Open AND WB_L.State = 0) THEN WB_L.B_Open := TRUE; Init := FALSE; END_IF

		IF Init THEN
			WB_A.B_Open := FALSE;
			WB_E.B_Open := FALSE;
			WB_K.B_Open := FALSE;
			WB_L.B_Open := FALSE;

			TimeCnt  := 0.0;

			IF SF_S_Fwd THEN
				TimeCnt := 0.0;
				State   := 5000;
				Next    := 0;
			ELSE
				EVP_Pump := REAL_TO_INT(EVP_Pump_Tgt * Perc * 10.0);
				OUT_LP   := 1;
				State    := State + 100; (*Port Fwd Dump - Pump*)
			END_IF

		END_IF
	END_IF

(*Port Aft Move - Open Valves3*)
3520:
	IF Manual OR NOT Ready THEN
		State := 0;

	ELSIF TimeCnt > CFG.TimeMax_Init THEN
		Error := State;
		State := 0;

	ELSIF Event_Stop = INIT_CONTINUOUS OR Event_Dump = INIT_CONTINUOUS OR Event_Fill = INIT_CONTINUOUS THEN
		WB_D.B_Open := FALSE;
		WB_E.B_Open := FALSE;
		WB_M.B_Open := FALSE;
		WB_L.B_Open := FALSE;

		TimeCnt := 0.0;
		State   := 5000;
		Next    := 0;

	ELSE
		IF Event_Move = INIT_CONTINUOUS THEN
			Pause := NOT Pause;
		END_IF

		Init := TRUE;
		IF NOT (WB_D.SF_Open AND WB_D.State = 0) THEN WB_D.B_Open := TRUE; Init := FALSE; END_IF
		IF NOT (WB_E.SF_Open AND WB_E.State = 0) THEN WB_E.B_Open := TRUE; Init := FALSE; END_IF
		IF NOT (WB_M.SF_Open AND WB_M.State = 0) THEN WB_M.B_Open := TRUE; Init := FALSE; END_IF
		IF NOT (WB_L.SF_Open AND WB_L.State = 0) THEN WB_L.B_Open := TRUE; Init := FALSE; END_IF

		IF Init THEN
			WB_D.B_Open := FALSE;
			WB_E.B_Open := FALSE;
			WB_M.B_Open := FALSE;
			WB_L.B_Open := FALSE;

			TimeCnt  := 0.0;

			IF SF_S_Aft THEN
				TimeCnt := 0.0;
				State   := 5000;
				Next    := 0;
			ELSE
				EVP_Pump := REAL_TO_INT(EVP_Pump_Tgt * Perc * 10.0);
				OUT_LP   := 1;
				State    := State + 100; (*Port Fwd Dump - Pump*)
			END_IF

		END_IF
	END_IF

(*Stbd Fwd Move - Open Valves3*)
3530:
	IF Manual OR NOT Ready THEN
		State := 0;

	ELSIF TimeCnt > CFG.TimeMax_Init THEN
		Error := State;
		State := 0;

	ELSIF Event_Stop = INIT_CONTINUOUS OR Event_Dump = INIT_CONTINUOUS OR Event_Fill = INIT_CONTINUOUS THEN
		WB_A.B_Open := FALSE;
		WB_F.B_Open := FALSE;
		WB_H.B_Open := FALSE;
		WB_K.B_Open := FALSE;

		TimeCnt := 0.0;
		State   := 5000;
		Next    := 0;

	ELSE
		IF Event_Move = INIT_CONTINUOUS THEN
			Pause := NOT Pause;
		END_IF

		Init := TRUE;

		IF NOT (WB_A.SF_Open AND WB_A.State = 0) THEN WB_A.B_Open := TRUE; Init := FALSE; END_IF
		IF NOT (WB_F.SF_Open AND WB_F.State = 0) THEN WB_F.B_Open := TRUE; Init := FALSE; END_IF
		IF NOT (WB_H.SF_Open AND WB_H.State = 0) THEN WB_H.B_Open := TRUE; Init := FALSE; END_IF
		IF NOT (WB_K.SF_Open AND WB_K.State = 0) THEN WB_K.B_Open := TRUE; Init := FALSE; END_IF

		IF Init THEN
			WB_A.B_Open := FALSE;
			WB_F.B_Open := FALSE;
			WB_H.B_Open := FALSE;
			WB_K.B_Open := FALSE;

			TimeCnt  := 0.0;

			IF SF_P_Fwd THEN
				TimeCnt := 0.0;
				State   := 5000;
				Next    := 0;
			ELSE
				EVP_Pump := REAL_TO_INT(EVP_Pump_Tgt * Perc * 10.0);
				OUT_LP   := 1;
				State    := State + 100; (*Port Fwd Dump - Pump*)
			END_IF

		END_IF
	END_IF

(*Stbd Aft Move - Open Valves3*)
3540:
	IF Manual OR NOT Ready THEN
		State := 0;

	ELSIF TimeCnt > CFG.TimeMax_Init THEN
		Error := State;
		State := 0;

	ELSIF Event_Stop = INIT_CONTINUOUS OR Event_Dump = INIT_CONTINUOUS OR Event_Fill = INIT_CONTINUOUS THEN
		WB_D.B_Open := FALSE;
		WB_F.B_Open := FALSE;
		WB_H.B_Open := FALSE;
		WB_M.B_Open := FALSE;

		TimeCnt := 0.0;
		State   := 5000;
		Next    := 0;

	ELSE
		IF Event_Move = INIT_CONTINUOUS THEN
			Pause := NOT Pause;
		END_IF

		Init := TRUE;

		IF NOT (WB_D.SF_Open AND WB_D.State = 0) THEN WB_D.B_Open := TRUE; Init := FALSE; END_IF
		IF NOT (WB_F.SF_Open AND WB_F.State = 0) THEN WB_F.B_Open := TRUE; Init := FALSE; END_IF
		IF NOT (WB_H.SF_Open AND WB_H.State = 0) THEN WB_H.B_Open := TRUE; Init := FALSE; END_IF
		IF NOT (WB_M.SF_Open AND WB_M.State = 0) THEN WB_M.B_Open := TRUE; Init := FALSE; END_IF

		IF Init THEN
			WB_D.B_Open := FALSE;
			WB_F.B_Open := FALSE;
			WB_H.B_Open := FALSE;
			WB_M.B_Open := FALSE;

			TimeCnt  := 0.0;

			IF SF_P_Aft THEN
				TimeCnt := 0.0;
				State   := 5000;
				Next    := 0;
			ELSE
				EVP_Pump := REAL_TO_INT(EVP_Pump_Tgt * Perc * 10.0);
				OUT_LP   := 1;
				State    := State + 100; (*Port Fwd Dump - Pump*)
			END_IF

		END_IF
	END_IF

(*Move Pump*)
3610,3620,3630,3640:
	IF Manual OR NOT Ready THEN
		OUT_LP   := 0;
		State    := 0;

	ELSE
		IF Event_Stop = INIT_CONTINUOUS OR Event_Fill = INIT_CONTINUOUS OR Event_Move = INIT_CONTINUOUS
		OR State = 3610 AND SF_S_Fwd
		OR State = 3620 AND SF_S_Aft
		OR State = 3630 AND SF_P_Fwd
		OR State = 3640 AND SF_P_Aft
		THEN
			SoftStop := TRUE;
		END_IF

		IF Event_Move = INIT_CONTINUOUS THEN
			Pause := NOT Pause;
		END_IF

		IF SoftStop OR Pause THEN
			EVP_Pump_Tgt := EVP_Pump_Tgt - CFG.EVP_Pump_Dec * CFG.Cycle;
			EVP_Pump_Tgt := MIN(EVP_Pump_Tgt, CFG.EVP_Pump_Max);
			EVP_Pump_Tgt := MAX(EVP_Pump_Tgt, CFG.EVP_Pump_Min);

			IF EVP_Pump_Tgt = CFG.EVP_Pump_Min OR CFG.EVP_Pump_Dec <= 0
			THEN EVP_Pump := 0;
			ELSE EVP_Pump := REAL_TO_UINT(EVP_Pump_Tgt * Perc * 10.0);
			END_IF

		ELSE
			EVP_Pump_Tgt := EVP_Pump_Tgt + CFG.EVP_Pump_Inc * CFG.Cycle;
			EVP_Pump_Tgt := MIN(EVP_Pump_Tgt, CFG.EVP_Pump_Max);
			EVP_Pump_Tgt := MAX(EVP_Pump_Tgt, CFG.EVP_Pump_Min);

			EVP_Pump := REAL_TO_UINT(EVP_Pump_Tgt * Perc * 10.0);

		END_IF

		IF EVP_Pump = 0 THEN
			OUT_LP := 0;

			IF SoftStop THEN
				TimeCnt := 0.0;
				State   := 5000;
				Next    := 0;
			END_IF

		ELSE
			OUT_LP := 1;

		END_IF
	END_IF


(*****************************************************************************)
(** INIT                                                                    **)
(*****************************************************************************)
(*Init Status - Valves*)
5000:
	OUT_Stop := TRUE;

	IF Manual OR NOT Ready THEN
		State := 0;

	ELSIF TimeCnt > CFG.TimeMax_Init THEN
		TimeCnt := 0.0;
		Error   := State;
		State   := 5001; (*Siempre fuerzo el scoop*)

	ELSE
		Init := TRUE;
	
		IF NOT (WB_A.SF_Close AND WB_A.State = 0) THEN WB_A.B_Close := TRUE; Init := FALSE; END_IF
		IF NOT (WB_B.SF_Close AND WB_B.State = 0) THEN WB_B.B_Close := TRUE; Init := FALSE; END_IF
		IF NOT (WB_C.SF_Close AND WB_C.State = 0) THEN WB_C.B_Close := TRUE; Init := FALSE; END_IF
		IF NOT (WB_D.SF_Close AND WB_D.State = 0) THEN WB_D.B_Close := TRUE; Init := FALSE; END_IF
		IF NOT (WB_E.SF_Close AND WB_E.State = 0) THEN WB_E.B_Close := TRUE; Init := FALSE; END_IF
		IF NOT (WB_F.SF_Close AND WB_F.State = 0) THEN WB_F.B_Close := TRUE; Init := FALSE; END_IF
		IF NOT (WB_G.SF_Close AND WB_G.State = 0) THEN WB_G.B_Close := TRUE; Init := FALSE; END_IF
		IF NOT (WB_H.SF_Close AND WB_H.State = 0) THEN WB_H.B_Close := TRUE; Init := FALSE; END_IF
		IF NOT (WB_I.SF_Close AND WB_I.State = 0) THEN WB_I.B_Close := TRUE; Init := FALSE; END_IF
		IF NOT (WB_J.SF_Close AND WB_J.State = 0) THEN WB_J.B_Close := TRUE; Init := FALSE; END_IF
		IF NOT (WB_K.SF_Close AND WB_K.State = 0) THEN WB_K.B_Close := TRUE; Init := FALSE; END_IF
		IF NOT (WB_L.SF_Close AND WB_L.State = 0) THEN WB_L.B_Close := TRUE; Init := FALSE; END_IF
		IF NOT (WB_M.SF_Close AND WB_M.State = 0) THEN WB_M.B_Close := TRUE; Init := FALSE; END_IF
		IF NOT (WB_N.SF_Close AND WB_N.State = 0) THEN WB_N.B_Close := TRUE; Init := FALSE; END_IF
		IF NOT (WB_R.SF_Close AND WB_R.State = 0) THEN WB_R.B_Close := TRUE; Init := FALSE; END_IF
		IF NOT (WB_S.SF_Close AND WB_S.State = 0) THEN WB_S.B_Close := TRUE; Init := FALSE; END_IF

		IF Init THEN
			WB_A.B_Close := FALSE;
			WB_B.B_Close := FALSE;
			WB_C.B_Close := FALSE;
			WB_D.B_Close := FALSE;
			WB_E.B_Close := FALSE;
			WB_F.B_Close := FALSE;
			WB_G.B_Close := FALSE;
			WB_H.B_Close := FALSE;
			WB_I.B_Close := FALSE;
			WB_J.B_Close := FALSE;
			WB_K.B_Close := FALSE;
			WB_L.B_Close := FALSE;
			WB_M.B_Close := FALSE;
			WB_N.B_Close := FALSE;
			WB_R.B_Close := FALSE;
			WB_S.B_Close := FALSE;

			State := 5001;

		END_IF
	END_IF

(*Init Status - Scoop UP*)
5001:
	IF Manual OR NOT Ready THEN
		State := 0;

	ELSIF TimeCnt > CFG.TimeMax_Init THEN
		Error := State;
		State := 0;

	ELSE
		Init := TRUE;
	
		IF NOT (WB_PUD.SF_Close AND WB_PUD.State = 0) THEN WB_PUD.B_Close := TRUE; Init := FALSE; END_IF
		IF NOT (WB_SUD.SF_Close AND WB_SUD.State = 0) THEN WB_SUD.B_Close := TRUE; Init := FALSE; END_IF

		IF CFG.EnScoopAF THEN
			IF NOT (WB_PAF.SF_Close AND WB_PAF.State = 0) THEN WB_PAF.B_Close := TRUE; Init := FALSE; END_IF (*test1*)
			IF NOT (WB_SAF.SF_Close AND WB_SAF.State = 0) THEN WB_SAF.B_Close := TRUE; Init := FALSE; END_IF (*test2*)
		END_IF

		IF Init THEN
			WB_PUD.B_Close := FALSE;
			WB_SUD.B_Close := FALSE;

			WB_PAF.B_Close := FALSE; (*test3*)
			WB_SAF.B_Close := FALSE; (*test4*)

			TimeCnt := 0.0;	 (*test5*)
			State   := Next; (*test6*)

			IF State = 0 THEN
				OUT_P_Fwd := FALSE;
				OUT_P_Aft := FALSE;
				OUT_S_Fwd := FALSE;
				OUT_S_Aft := FALSE;
				OUT_12    := FALSE;
			END_IF

			(*State := 5002;*) (*test7*)

		END_IF
	END_IF

(*Init Status - Scoop FWD*) (*No enta mas!*)
(*5002:
	IF Manual OR NOT Ready THEN
		State := 0;

	ELSIF TimeCnt > CFG.TimeMax_Init THEN
		Error := State;
		State := 0;

	ELSE
		Init := TRUE;
	
		IF NOT (WB_PAF.SF_Close AND WB_PAF.State = 0) THEN WB_PAF.B_Close := TRUE; Init := FALSE; END_IF
		IF NOT (WB_SAF.SF_Close AND WB_SAF.State = 0) THEN WB_SAF.B_Close := TRUE; Init := FALSE; END_IF

		IF Init THEN
			WB_PAF.B_Close := FALSE;
			WB_SAF.B_Close := FALSE;

			TimeCnt := 0.0;
			State   := Next;

		END_IF
	END_IF*)

END_CASE

OUT_Pump := EVP_Pump <> 0;

(*
	PAF y SAF disabled
*)



(*Recordar PUMP EV1608 multiplicar por 10.0*)

(*	IF NOT (WB_A.SF_Close AND WB_A.State = 0) THEN WB_A.B_Close := TRUE; Init := FALSE; END_IF
	IF NOT (WB_B.SF_Close AND WB_B.State = 0) THEN WB_B.B_Close := TRUE; Init := FALSE; END_IF
	IF NOT (WB_C.SF_Close AND WB_C.State = 0) THEN WB_C.B_Close := TRUE; Init := FALSE; END_IF
	IF NOT (WB_D.SF_Close AND WB_D.State = 0) THEN WB_D.B_Close := TRUE; Init := FALSE; END_IF
	IF NOT (WB_E.SF_Close AND WB_E.State = 0) THEN WB_E.B_Close := TRUE; Init := FALSE; END_IF
	IF NOT (WB_F.SF_Close AND WB_F.State = 0) THEN WB_F.B_Close := TRUE; Init := FALSE; END_IF
	IF NOT (WB_G.SF_Close AND WB_G.State = 0) THEN WB_G.B_Close := TRUE; Init := FALSE; END_IF
	IF NOT (WB_H.SF_Close AND WB_H.State = 0) THEN WB_H.B_Close := TRUE; Init := FALSE; END_IF
	IF NOT (WB_I.SF_Close AND WB_I.State = 0) THEN WB_I.B_Close := TRUE; Init := FALSE; END_IF
	IF NOT (WB_J.SF_Close AND WB_J.State = 0) THEN WB_J.B_Close := TRUE; Init := FALSE; END_IF
	IF NOT (WB_K.SF_Close AND WB_K.State = 0) THEN WB_K.B_Close := TRUE; Init := FALSE; END_IF
	IF NOT (WB_L.SF_Close AND WB_L.State = 0) THEN WB_L.B_Close := TRUE; Init := FALSE; END_IF
	IF NOT (WB_M.SF_Close AND WB_M.State = 0) THEN WB_M.B_Close := TRUE; Init := FALSE; END_IF
	IF NOT (WB_N.SF_Close AND WB_N.State = 0) THEN WB_N.B_Close := TRUE; Init := FALSE; END_IF
	IF NOT (WB_R.SF_Close AND WB_R.State = 0) THEN WB_R.B_Close := TRUE; Init := FALSE; END_IF
	IF NOT (WB_S.SF_Close AND WB_S.State = 0) THEN WB_S.B_Close := TRUE; Init := FALSE; END_IF

